Yaskawa INFORM job: apremTRJ1.JBI

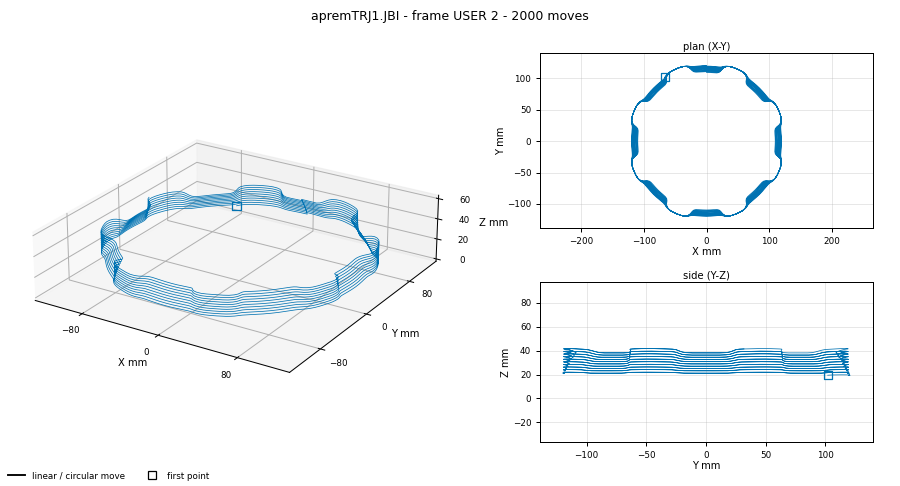
[picture p0: tool path of apremTRJ1.JBI in frame USER 2, 2000 of 2000 moves have a stored position in this frame; points joined in program order, loops and branches not executed]
/JOB
//NAME apremTRJ1
//POS
///NPOS 2000,0,0,0,0,0
///USER 2
///TOOL 1
///POSTYPE USER
///RECTAN
///RCONF 1,0,0,0,0,0,0,0,0,0,0,0,0,0,0,0,0,0,0,0,0,0,0,0
C00000=-66.629,101.942,19.455,-170.1157,12.4530,0.0000
C00001=-65.347,103.638,19.586,-173.5152,9.1234,0.0000
C00002=-64.038,105.345,19.680,-175.2675,5.6483,0.0000
C00003=-62.177,107.232,19.725,-176.7314,2.8984,0.0000
C00004=-59.447,109.388,19.749,-178.4360,1.1171,0.0000
C00005=-56.168,111.510,19.767,-179.6465,0.2072,0.0000
C00006=-52.762,113.295,19.786,-179.9247,0.0358,0.0000
C00007=-49.468,114.792,19.798,-179.9913,0.0038,0.0000
C00008=-46.191,116.149,19.798,-179.9912,0.0035,0.0000
C00009=-42.803,117.420,19.786,-179.9215,0.0280,0.0000
C00010=-39.133,118.567,19.767,-179.6035,0.1035,0.0000
C00011=-35.314,119.384,19.749,-178.1045,0.3162,0.0000
C00012=-31.859,119.791,19.725,-175.6434,0.2625,0.0000
C00013=-29.209,119.772,19.680,-172.6791,-0.6529,0.0000
C00014=-27.076,119.491,19.586,-169.0248,-1.9005,0.0000
C00015=-24.970,119.198,19.455,-164.3916,-1.8868,0.0000
C00016=-22.390,119.093,19.319,-160.1217,-0.0530,0.0000
C00017=-18.637,119.331,19.213,-157.6149,2.1562,0.0000
C00018=-13.062,119.916,19.170,-156.7679,2.4486,0.0000
C00019=-6.840,120.423,19.168,-156.6463,1.4246,0.0000
C00020=0.000,120.619,19.169,-156.6224,0.0002,0.0000
C00021=0.000,119.715,21.175,-154.8867,0.0002,0.0000
C00022=6.757,119.522,21.173,-154.9119,-1.5414,0.0000
C00023=12.923,119.024,21.176,-155.0380,-2.5924,0.0000
C00024=18.467,118.472,21.232,-155.9401,-1.9735,0.0000
C00025=22.185,118.320,21.368,-158.8454,1.0092,0.0000
C00026=24.738,118.553,21.546,-163.9075,3.1512,0.0000
C00027=26.827,119.004,21.717,-169.0787,2.8689,0.0000
C00028=28.944,119.457,21.842,-172.7347,1.2029,0.0000
C00029=31.572,119.635,21.901,-175.6219,-0.0566,0.0000
C00030=35.044,119.351,21.932,-178.1277,-0.2593,0.0000
C00031=38.919,118.606,21.957,-179.6493,-0.0862,0.0000
C00032=42.669,117.464,21.982,-179.9232,-0.0272,0.0000
C00033=46.146,116.167,21.998,-179.9915,-0.0033,0.0000
C00034=49.513,114.773,21.998,-179.9916,-0.0037,0.0000
C00035=52.889,113.231,21.982,-179.9265,-0.0351,0.0000
C00036=56.347,111.387,21.957,-179.6910,-0.1870,0.0000
C00037=59.614,109.174,21.932,-178.4926,-1.1409,0.0000
C00038=62.270,106.919,21.901,-176.8613,-3.0589,0.0000
C00039=64.002,104.935,21.842,-175.6938,-5.9938,0.0000
C00040=65.179,103.118,21.717,-174.2325,-9.7524,0.0000
C00041=66.337,101.322,21.546,-170.6269,-13.6541,0.0000
C00042=67.977,99.352,21.368,-165.3631,-15.9648,0.0000
C00043=70.714,96.831,21.232,-161.2181,-16.2433,0.0000
C00044=75.024,93.301,21.176,-160.1416,-16.5489,0.0000
C00045=79.737,89.293,21.173,-160.7058,-17.3293,0.0000
C00046=84.652,84.652,21.175,-161.6632,-18.3371,0.0000
C00047=89.293,79.737,21.173,-162.6706,-19.2941,0.0000
C00048=93.301,75.024,21.176,-163.4508,-19.8582,0.0000
C00049=96.831,70.714,21.232,-163.7569,-18.7820,0.0000
C00050=99.352,67.977,21.368,-164.0352,-14.6369,0.0000
C00051=101.322,66.337,21.546,-166.3459,-9.3731,0.0000
C00052=103.118,65.179,21.717,-170.2476,-5.7675,0.0000
C00053=104.935,64.002,21.842,-174.0062,-4.3062,0.0000
C00054=106.919,62.270,21.901,-176.9411,-3.1387,0.0000
C00055=109.174,59.614,21.932,-178.8591,-1.5074,0.0000
C00056=111.387,56.347,21.957,-179.8130,-0.3090,0.0000
C00057=113.231,52.889,21.982,-179.9649,-0.0735,0.0000
C00058=114.773,49.513,21.998,-179.9963,-0.0084,0.0000
C00059=116.167,46.146,21.998,-179.9967,-0.0085,0.0000
C00060=117.464,42.669,21.982,-179.9728,-0.0768,0.0000
C00061=118.606,38.919,21.957,-179.9138,-0.3507,0.0000
C00062=119.351,35.044,21.932,-179.7407,-1.8723,0.0000
C00063=119.635,31.572,21.901,-179.9434,-4.3781,0.0000
C00064=119.457,28.944,21.842,178.7971,-7.2653,0.0000
C00065=119.004,26.827,21.717,177.1311,-10.9213,0.0000
C00066=118.553,24.738,21.546,176.8488,-16.0925,0.0000
C00067=118.320,22.185,21.368,178.9908,-21.1546,0.0000
C00068=118.472,18.467,21.232,-178.0265,-24.0599,0.0000
C00069=119.024,12.923,21.176,-177.4076,-24.9620,0.0000
C00070=119.522,6.757,21.173,-178.4586,-25.0881,0.0000
C00071=119.715,0.000,21.175,179.9998,-25.1133,0.0000
C00072=119.522,-6.757,21.173,178.4588,-25.0881,0.0000
C00073=119.024,-12.923,21.176,177.4079,-24.9620,0.0000
C00074=118.472,-18.468,21.232,178.0263,-24.0599,0.0000
C00075=118.320,-22.185,21.368,-178.9908,-21.1546,0.0000
C00076=118.553,-24.738,21.546,-176.8488,-16.0925,0.0000
C00077=119.004,-26.827,21.717,-177.1311,-10.9213,0.0000
C00078=119.457,-28.944,21.842,-178.7971,-7.2653,0.0000
C00079=119.635,-31.572,21.901,179.9434,-4.3781,0.0000
C00080=119.351,-35.044,21.932,179.7407,-1.8723,0.0000
C00081=118.606,-38.919,21.957,179.9138,-0.3507,0.0000
C00082=117.464,-42.669,21.982,179.9728,-0.0768,0.0000
C00083=116.167,-46.146,21.998,179.9967,-0.0085,0.0000
C00084=114.773,-49.513,21.998,179.9963,-0.0084,0.0000
C00085=113.231,-52.889,21.982,179.9649,-0.0735,0.0000
C00086=111.387,-56.347,21.957,179.8130,-0.3090,0.0000
C00087=109.174,-59.614,21.932,178.8591,-1.5074,0.0000
C00088=106.919,-62.270,21.901,176.9411,-3.1387,0.0000
C00089=104.935,-64.002,21.842,174.0062,-4.3062,0.0000
C00090=103.118,-65.179,21.717,170.2476,-5.7675,0.0000
C00091=101.322,-66.337,21.546,166.3459,-9.3731,0.0000
C00092=99.352,-67.977,21.368,164.0352,-14.6369,0.0000
C00093=96.831,-70.714,21.232,163.7567,-18.7819,0.0000
C00094=93.301,-75.024,21.176,163.4511,-19.8584,0.0000
C00095=89.293,-79.737,21.173,162.6707,-19.2942,0.0000
C00096=84.652,-84.652,21.175,161.6629,-18.3368,0.0000
C00097=79.737,-89.293,21.173,160.7059,-17.3294,0.0000
C00098=75.024,-93.301,21.176,160.1418,-16.5492,0.0000
C00099=70.714,-96.831,21.232,161.2180,-16.2431,0.0000
C00100=67.977,-99.352,21.368,165.3631,-15.9648,0.0000
C00101=66.337,-101.322,21.546,170.6269,-13.6541,0.0000
C00102=65.179,-103.118,21.717,174.2325,-9.7524,0.0000
C00103=64.002,-104.935,21.842,175.6938,-5.9938,0.0000
C00104=62.270,-106.919,21.901,176.8613,-3.0589,0.0000
C00105=59.614,-109.174,21.932,178.4926,-1.1409,0.0000
C00106=56.347,-111.387,21.957,179.6910,-0.1870,0.0000
C00107=52.889,-113.231,21.982,179.9265,-0.0351,0.0000
C00108=49.513,-114.773,21.998,179.9916,-0.0037,0.0000
C00109=46.146,-116.167,21.998,179.9915,-0.0033,0.0000
C00110=42.669,-117.464,21.982,179.9232,-0.0272,0.0000
C00111=38.919,-118.606,21.957,179.6493,-0.0862,0.0000
C00112=35.044,-119.351,21.932,178.1277,-0.2593,0.0000
C00113=31.572,-119.635,21.901,175.6219,-0.0566,0.0000
C00114=28.944,-119.457,21.842,172.7347,1.2029,0.0000
C00115=26.827,-119.004,21.717,169.0787,2.8689,0.0000
C00116=24.738,-118.553,21.546,163.9075,3.1512,0.0000
C00117=22.185,-118.320,21.368,158.8454,1.0092,0.0000
C00118=18.467,-118.472,21.232,155.9401,-1.9735,0.0000
C00119=12.923,-119.024,21.176,155.0380,-2.5924,0.0000
C00120=6.757,-119.522,21.173,154.9119,-1.5414,0.0000
C00121=0.000,-119.715,21.175,154.8867,0.0002,0.0000
C00122=0.000,-119.715,21.175,154.8867,0.0002,0.0000
C00123=-6.757,-119.522,21.173,154.9119,1.5412,0.0000
C00124=-12.923,-119.024,21.176,155.0380,2.5921,0.0000
C00125=-18.468,-118.472,21.232,155.9401,1.9737,0.0000
C00126=-22.185,-118.320,21.368,158.8454,-1.0092,0.0000
C00127=-24.738,-118.553,21.546,163.9075,-3.1512,0.0000
C00128=-26.827,-119.004,21.717,169.0787,-2.8689,0.0000
C00129=-28.944,-119.457,21.842,172.7347,-1.2029,0.0000
C00130=-31.572,-119.635,21.901,175.6219,0.0566,0.0000
C00131=-35.044,-119.351,21.932,178.1277,0.2593,0.0000
C00132=-38.919,-118.606,21.957,179.6493,0.0862,0.0000
C00133=-42.669,-117.464,21.982,179.9232,0.0272,0.0000
C00134=-46.146,-116.167,21.998,179.9915,0.0033,0.0000
C00135=-49.513,-114.773,21.998,179.9916,0.0037,0.0000
C00136=-52.889,-113.231,21.982,179.9265,0.0351,0.0000
C00137=-56.347,-111.387,21.957,179.6910,0.1870,0.0000
C00138=-59.614,-109.174,21.932,178.4926,1.1409,0.0000
C00139=-62.270,-106.919,21.901,176.8613,3.0589,0.0000
C00140=-64.002,-104.935,21.842,175.6938,5.9938,0.0000
C00141=-65.179,-103.118,21.717,174.2325,9.7524,0.0000
C00142=-66.337,-101.322,21.546,170.6269,13.6541,0.0000
C00143=-67.977,-99.352,21.368,165.3631,15.9648,0.0000
C00144=-70.714,-96.831,21.232,161.2181,16.2433,0.0000
C00145=-75.024,-93.301,21.176,160.1416,16.5489,0.0000
C00146=-79.737,-89.293,21.173,160.7058,17.3293,0.0000
C00147=-84.652,-84.652,21.175,161.6632,18.3371,0.0000
C00148=-89.293,-79.737,21.173,162.6706,19.2941,0.0000
C00149=-93.301,-75.024,21.176,163.4508,19.8582,0.0000
C00150=-96.831,-70.714,21.232,163.7569,18.7820,0.0000
C00151=-99.352,-67.977,21.368,164.0352,14.6369,0.0000
C00152=-101.322,-66.337,21.546,166.3459,9.3731,0.0000
C00153=-103.118,-65.179,21.717,170.2476,5.7675,0.0000
C00154=-104.935,-64.002,21.842,174.0062,4.3062,0.0000
C00155=-106.919,-62.270,21.901,176.9411,3.1387,0.0000
C00156=-109.174,-59.614,21.932,178.8591,1.5074,0.0000
C00157=-111.387,-56.347,21.957,179.8130,0.3090,0.0000
C00158=-113.231,-52.889,21.982,179.9649,0.0735,0.0000
C00159=-114.773,-49.513,21.998,179.9963,0.0084,0.0000
C00160=-116.167,-46.146,21.998,179.9967,0.0085,0.0000
C00161=-117.464,-42.669,21.982,179.9728,0.0768,0.0000
C00162=-118.606,-38.919,21.957,179.9138,0.3507,0.0000
C00163=-119.351,-35.044,21.932,179.7407,1.8723,0.0000
C00164=-119.635,-31.572,21.901,179.9434,4.3781,0.0000
C00165=-119.457,-28.944,21.842,-178.7971,7.2653,0.0000
C00166=-119.004,-26.827,21.717,-177.1311,10.9213,0.0000
C00167=-118.553,-24.738,21.546,-176.8488,16.0925,0.0000
C00168=-118.320,-22.185,21.368,-178.9908,21.1546,0.0000
C00169=-118.472,-18.467,21.232,178.0265,24.0599,0.0000
C00170=-119.024,-12.923,21.176,177.4076,24.9620,0.0000
C00171=-119.522,-6.757,21.173,178.4586,25.0881,0.0000
C00172=-119.715,0.000,21.175,-179.9998,25.1133,0.0000
C00173=-119.522,6.757,21.173,-178.4588,25.0881,0.0000
C00174=-119.024,12.923,21.176,-177.4079,24.9620,0.0000
C00175=-118.472,18.468,21.232,-178.0263,24.0599,0.0000
C00176=-118.320,22.185,21.368,178.9908,21.1546,0.0000
C00177=-118.553,24.738,21.546,176.8488,16.0925,0.0000
C00178=-119.004,26.827,21.717,177.1311,10.9213,0.0000
C00179=-119.457,28.944,21.842,178.7971,7.2653,0.0000
C00180=-119.635,31.572,21.901,-179.9434,4.3781,0.0000
C00181=-119.351,35.044,21.932,-179.7407,1.8723,0.0000
C00182=-118.606,38.919,21.957,-179.9138,0.3507,0.0000
C00183=-117.464,42.669,21.982,-179.9728,0.0768,0.0000
C00184=-116.167,46.146,21.998,-179.9967,0.0085,0.0000
C00185=-114.773,49.513,21.998,-179.9963,0.0084,0.0000
C00186=-113.231,52.889,21.982,-179.9649,0.0735,0.0000
C00187=-111.387,56.347,21.957,-179.8130,0.3090,0.0000
C00188=-109.174,59.614,21.932,-178.8591,1.5074,0.0000
C00189=-106.919,62.270,21.901,-176.9411,3.1387,0.0000
C00190=-104.935,64.002,21.842,-174.0062,4.3062,0.0000
C00191=-103.118,65.179,21.717,-170.2476,5.7675,0.0000
C00192=-101.322,66.337,21.546,-166.3459,9.3731,0.0000
C00193=-99.352,67.977,21.368,-164.0352,14.6369,0.0000
C00194=-96.831,70.714,21.232,-163.7567,18.7819,0.0000
C00195=-93.301,75.024,21.176,-163.4511,19.8584,0.0000
C00196=-89.293,79.737,21.173,-162.6707,19.2942,0.0000
C00197=-84.652,84.652,21.175,-161.6629,18.3368,0.0000
C00198=-79.737,89.293,21.173,-160.7059,17.3294,0.0000
C00199=-75.024,93.301,21.176,-160.1418,16.5492,0.0000
C00200=-70.714,96.831,21.232,-161.2180,16.2431,0.0000
C00201=-67.977,99.352,21.368,-165.3631,15.9648,0.0000
C00202=-66.337,101.322,21.546,-170.6269,13.6541,0.0000
C00203=-65.179,103.118,21.717,-174.2325,9.7524,0.0000
C00204=-64.002,104.935,21.842,-175.6938,5.9938,0.0000
C00205=-62.270,106.919,21.901,-176.8613,3.0589,0.0000
C00206=-59.614,109.174,21.932,-178.4926,1.1409,0.0000
C00207=-56.347,111.387,21.957,-179.6910,0.1870,0.0000
C00208=-52.889,113.231,21.982,-179.9265,0.0351,0.0000
C00209=-49.513,114.773,21.998,-179.9916,0.0037,0.0000
C00210=-46.146,116.167,21.998,-179.9915,0.0033,0.0000
C00211=-42.669,117.464,21.982,-179.9232,0.0272,0.0000
C00212=-38.919,118.606,21.957,-179.6493,0.0862,0.0000
C00213=-35.044,119.351,21.932,-178.1277,0.2593,0.0000
C00214=-31.572,119.635,21.901,-175.6219,0.0566,0.0000
C00215=-28.944,119.457,21.842,-172.7347,-1.2029,0.0000
C00216=-26.827,119.004,21.717,-169.0787,-2.8689,0.0000
C00217=-24.738,118.553,21.546,-163.9075,-3.1512,0.0000
C00218=-22.185,118.320,21.368,-158.8454,-1.0092,0.0000
C00219=-18.468,118.472,21.232,-155.9401,1.9737,0.0000
C00220=-12.923,119.024,21.176,-155.0380,2.5921,0.0000
C00221=-6.757,119.522,21.173,-154.9119,1.5412,0.0000
C00222=0.000,119.715,21.175,-154.8867,0.0002,0.0000
C00223=0.000,118.754,23.154,-153.2988,0.0002,0.0000
C00224=6.669,118.564,23.151,-153.3252,-1.6500,0.0000
C00225=12.776,118.074,23.155,-153.4547,-2.7089,0.0000
C00226=18.287,117.558,23.225,-154.4168,-1.6956,0.0000
C00227=21.966,117.495,23.396,-157.8261,2.1572,0.0000
C00228=24.490,117.863,23.620,-163.8200,4.4801,0.0000
C00229=26.560,118.482,23.837,-169.5033,3.7726,0.0000
C00230=28.658,119.117,23.996,-173.0515,1.7294,0.0000
C00231=31.262,119.466,24.073,-175.7313,0.1639,0.0000
C00232=34.753,119.316,24.112,-178.2061,-0.1949,0.0000
C00233=38.689,118.647,24.144,-179.7139,-0.0658,0.0000
C00234=42.523,117.512,24.176,-179.9268,-0.0257,0.0000
C00235=46.096,116.186,24.197,-179.9920,-0.0031,0.0000
C00236=49.561,114.751,24.197,-179.9921,-0.0034,0.0000
C00237=53.026,113.162,24.176,-179.9301,-0.0336,0.0000
C00238=56.539,111.253,24.144,-179.7511,-0.1558,0.0000
C00239=59.796,108.943,24.112,-178.5936,-1.1309,0.0000
C00240=62.370,106.581,24.073,-177.0944,-3.1368,0.0000
C00241=63.964,104.493,23.996,-176.2909,-6.1372,0.0000
C00242=64.998,102.560,23.837,-175.1764,-10.0729,0.0000
C00243=66.025,100.658,23.620,-171.4825,-14.6048,0.0000
C00244=67.549,98.614,23.396,-165.3424,-17.4753,0.0000
C00245=70.195,96.057,23.225,-160.2282,-17.6199,0.0000
C00246=74.457,92.525,23.155,-158.8582,-17.7339,0.0000
C00247=79.121,88.553,23.151,-159.4130,-18.5146,0.0000
C00248=83.972,83.972,23.154,-160.4219,-19.5784,0.0000
C00249=88.553,79.121,23.151,-161.4852,-20.5868,0.0000
C00250=92.525,74.457,23.155,-162.2659,-21.1415,0.0000
C00251=96.057,70.195,23.225,-162.3803,-19.7719,0.0000
C00252=98.614,67.549,23.396,-162.5247,-14.6576,0.0000
C00253=100.658,66.025,23.620,-165.3952,-8.5175,0.0000
C00254=102.560,64.998,23.837,-169.9271,-4.8236,0.0000
C00255=104.493,63.964,23.996,-173.8628,-3.7091,0.0000
C00256=106.581,62.370,24.073,-176.8632,-2.9056,0.0000
C00257=108.943,59.796,24.112,-178.8691,-1.4064,0.0000
C00258=111.253,56.539,24.144,-179.8442,-0.2489,0.0000
C00259=113.162,53.026,24.176,-179.9664,-0.0699,0.0000
C00260=114.751,49.561,24.197,-179.9966,-0.0079,0.0000
C00261=116.186,46.096,24.197,-179.9969,-0.0080,0.0000
C00262=117.512,42.523,24.176,-179.9743,-0.0732,0.0000
C00263=118.647,38.689,24.144,-179.9342,-0.2861,0.0000
C00264=119.316,34.753,24.112,-179.8051,-1.7939,0.0000
C00265=119.466,31.262,24.073,179.8361,-4.2687,0.0000
C00266=119.117,28.658,23.996,178.2706,-6.9485,0.0000
C00267=118.482,26.560,23.837,176.2274,-10.4967,0.0000
C00268=117.863,24.490,23.620,175.5199,-16.1800,0.0000
C00269=117.495,21.966,23.396,177.8428,-22.1739,0.0000
C00270=117.558,18.287,23.225,-178.3044,-25.5832,0.0000
C00271=118.074,12.776,23.155,-177.2911,-26.5453,0.0000
C00272=118.564,6.669,23.151,-178.3500,-26.6748,0.0000
C00273=118.754,0.000,23.154,179.9998,-26.7012,0.0000
C00274=118.564,-6.669,23.151,178.3503,-26.6748,0.0000
C00275=118.074,-12.776,23.155,177.2915,-26.5453,0.0000
C00276=117.558,-18.287,23.225,178.3041,-25.5831,0.0000
C00277=117.495,-21.966,23.396,-177.8428,-22.1739,0.0000
C00278=117.863,-24.490,23.620,-175.5199,-16.1800,0.0000
C00279=118.482,-26.560,23.837,-176.2274,-10.4967,0.0000
C00280=119.117,-28.658,23.996,-178.2706,-6.9485,0.0000
C00281=119.466,-31.262,24.073,-179.8361,-4.2687,0.0000
C00282=119.316,-34.753,24.112,179.8051,-1.7939,0.0000
C00283=118.647,-38.689,24.144,179.9342,-0.2861,0.0000
C00284=117.512,-42.523,24.176,179.9743,-0.0732,0.0000
C00285=116.186,-46.096,24.197,179.9969,-0.0080,0.0000
C00286=114.751,-49.561,24.197,179.9966,-0.0079,0.0000
C00287=113.162,-53.026,24.176,179.9664,-0.0699,0.0000
C00288=111.253,-56.539,24.144,179.8442,-0.2489,0.0000
C00289=108.943,-59.796,24.112,178.8691,-1.4064,0.0000
C00290=106.581,-62.370,24.073,176.8632,-2.9056,0.0000
C00291=104.493,-63.964,23.996,173.8628,-3.7091,0.0000
C00292=102.560,-64.998,23.837,169.9271,-4.8236,0.0000
C00293=100.658,-66.025,23.620,165.3952,-8.5175,0.0000
C00294=98.614,-67.549,23.396,162.5247,-14.6576,0.0000
C00295=96.057,-70.195,23.225,162.3801,-19.7718,0.0000
C00296=92.525,-74.457,23.155,162.2661,-21.1418,0.0000
C00297=88.553,-79.121,23.151,161.4854,-20.5870,0.0000
C00298=83.972,-83.972,23.154,160.4216,-19.5781,0.0000
C00299=79.121,-88.553,23.151,159.4132,-18.5148,0.0000
C00300=74.457,-92.525,23.155,158.8585,-17.7341,0.0000
C00301=70.195,-96.057,23.225,160.2281,-17.6197,0.0000
C00302=67.549,-98.614,23.396,165.3424,-17.4753,0.0000
C00303=66.025,-100.658,23.620,171.4825,-14.6048,0.0000
C00304=64.998,-102.560,23.837,175.1764,-10.0729,0.0000
C00305=63.964,-104.493,23.996,176.2909,-6.1372,0.0000
C00306=62.370,-106.581,24.073,177.0944,-3.1368,0.0000
C00307=59.796,-108.943,24.112,178.5936,-1.1309,0.0000
C00308=56.539,-111.253,24.144,179.7511,-0.1558,0.0000
C00309=53.026,-113.162,24.176,179.9301,-0.0336,0.0000
C00310=49.561,-114.751,24.197,179.9921,-0.0034,0.0000
C00311=46.096,-116.186,24.197,179.9920,-0.0031,0.0000
C00312=42.523,-117.512,24.176,179.9268,-0.0257,0.0000
C00313=38.689,-118.647,24.144,179.7139,-0.0658,0.0000
C00314=34.753,-119.316,24.112,178.2061,-0.1949,0.0000
C00315=31.262,-119.466,24.073,175.7313,0.1639,0.0000
C00316=28.658,-119.117,23.996,173.0515,1.7294,0.0000
C00317=26.560,-118.482,23.837,169.5033,3.7726,0.0000
C00318=24.490,-117.863,23.620,163.8200,4.4801,0.0000
C00319=21.966,-117.495,23.396,157.8261,2.1572,0.0000
C00320=18.287,-117.558,23.225,154.4168,-1.6956,0.0000
C00321=12.776,-118.074,23.155,153.4547,-2.7089,0.0000
C00322=6.669,-118.564,23.151,153.3252,-1.6500,0.0000
C00323=0.000,-118.754,23.154,153.2988,0.0002,0.0000
C00324=0.000,-118.754,23.154,153.2988,0.0002,0.0000
C00325=-6.669,-118.564,23.151,153.3252,1.6497,0.0000
C00326=-12.776,-118.074,23.155,153.4547,2.7085,0.0000
C00327=-18.287,-117.558,23.225,154.4169,1.6959,0.0000
C00328=-21.966,-117.495,23.396,157.8261,-2.1572,0.0000
C00329=-24.490,-117.863,23.620,163.8200,-4.4801,0.0000
C00330=-26.560,-118.482,23.837,169.5033,-3.7726,0.0000
C00331=-28.658,-119.117,23.996,173.0515,-1.7294,0.0000
C00332=-31.262,-119.466,24.073,175.7313,-0.1639,0.0000
C00333=-34.753,-119.316,24.112,178.2061,0.1949,0.0000
C00334=-38.689,-118.647,24.144,179.7139,0.0658,0.0000
C00335=-42.523,-117.512,24.176,179.9268,0.0257,0.0000
C00336=-46.096,-116.186,24.197,179.9920,0.0031,0.0000
C00337=-49.561,-114.751,24.197,179.9921,0.0034,0.0000
C00338=-53.026,-113.162,24.176,179.9301,0.0336,0.0000
C00339=-56.539,-111.253,24.144,179.7511,0.1558,0.0000
C00340=-59.796,-108.943,24.112,178.5936,1.1309,0.0000
C00341=-62.370,-106.581,24.073,177.0944,3.1368,0.0000
C00342=-63.964,-104.493,23.996,176.2909,6.1372,0.0000
C00343=-64.998,-102.560,23.837,175.1764,10.0729,0.0000
C00344=-66.025,-100.658,23.620,171.4825,14.6048,0.0000
C00345=-67.549,-98.614,23.396,165.3424,17.4753,0.0000
C00346=-70.195,-96.057,23.225,160.2282,17.6199,0.0000
C00347=-74.457,-92.525,23.155,158.8582,17.7339,0.0000
C00348=-79.121,-88.553,23.151,159.4130,18.5146,0.0000
C00349=-83.972,-83.972,23.154,160.4219,19.5784,0.0000
C00350=-88.553,-79.121,23.151,161.4852,20.5868,0.0000
C00351=-92.525,-74.457,23.155,162.2659,21.1415,0.0000
C00352=-96.057,-70.195,23.225,162.3803,19.7719,0.0000
C00353=-98.614,-67.549,23.396,162.5247,14.6576,0.0000
C00354=-100.658,-66.025,23.620,165.3952,8.5175,0.0000
C00355=-102.560,-64.998,23.837,169.9271,4.8236,0.0000
C00356=-104.493,-63.964,23.996,173.8628,3.7091,0.0000
C00357=-106.581,-62.370,24.073,176.8632,2.9056,0.0000
C00358=-108.943,-59.796,24.112,178.8691,1.4064,0.0000
C00359=-111.253,-56.539,24.144,179.8442,0.2489,0.0000
C00360=-113.162,-53.026,24.176,179.9664,0.0699,0.0000
C00361=-114.751,-49.561,24.197,179.9966,0.0079,0.0000
C00362=-116.186,-46.096,24.197,179.9969,0.0080,0.0000
C00363=-117.512,-42.523,24.176,179.9743,0.0732,0.0000
C00364=-118.647,-38.689,24.144,179.9342,0.2861,0.0000
C00365=-119.316,-34.753,24.112,179.8051,1.7939,0.0000
C00366=-119.466,-31.262,24.073,-179.8361,4.2687,0.0000
C00367=-119.117,-28.658,23.996,-178.2706,6.9485,0.0000
C00368=-118.482,-26.560,23.837,-176.2274,10.4967,0.0000
C00369=-117.863,-24.490,23.620,-175.5199,16.1800,0.0000
C00370=-117.495,-21.966,23.396,-177.8428,22.1739,0.0000
C00371=-117.558,-18.287,23.225,178.3044,25.5832,0.0000
C00372=-118.074,-12.776,23.155,177.2911,26.5453,0.0000
C00373=-118.564,-6.669,23.151,178.3500,26.6748,0.0000
C00374=-118.754,0.000,23.154,-179.9998,26.7012,0.0000
C00375=-118.564,6.669,23.151,-178.3503,26.6748,0.0000
C00376=-118.074,12.776,23.155,-177.2915,26.5453,0.0000
C00377=-117.558,18.287,23.225,-178.3041,25.5831,0.0000
C00378=-117.495,21.966,23.396,177.8428,22.1739,0.0000
C00379=-117.863,24.490,23.620,175.5199,16.1800,0.0000
C00380=-118.482,26.560,23.837,176.2274,10.4967,0.0000
C00381=-119.117,28.658,23.996,178.2706,6.9485,0.0000
C00382=-119.466,31.262,24.073,179.8361,4.2687,0.0000
C00383=-119.316,34.753,24.112,-179.8051,1.7939,0.0000
C00384=-118.647,38.689,24.144,-179.9342,0.2861,0.0000
C00385=-117.512,42.523,24.176,-179.9743,0.0732,0.0000
C00386=-116.186,46.096,24.197,-179.9969,0.0080,0.0000
C00387=-114.751,49.561,24.197,-179.9966,0.0079,0.0000
C00388=-113.162,53.026,24.176,-179.9664,0.0699,0.0000
C00389=-111.253,56.539,24.144,-179.8442,0.2489,0.0000
C00390=-108.943,59.796,24.112,-178.8691,1.4064,0.0000
C00391=-106.581,62.370,24.073,-176.8632,2.9056,0.0000
C00392=-104.493,63.964,23.996,-173.8628,3.7091,0.0000
C00393=-102.560,64.998,23.837,-169.9271,4.8236,0.0000
C00394=-100.658,66.025,23.620,-165.3952,8.5175,0.0000
C00395=-98.614,67.549,23.396,-162.5247,14.6576,0.0000
C00396=-96.057,70.195,23.225,-162.3801,19.7718,0.0000
C00397=-92.525,74.457,23.155,-162.2661,21.1418,0.0000
C00398=-88.553,79.121,23.151,-161.4854,20.5870,0.0000
C00399=-83.972,83.972,23.154,-160.4216,19.5781,0.0000
C00400=-79.121,88.553,23.151,-159.4132,18.5148,0.0000
C00401=-74.457,92.525,23.155,-158.8585,17.7341,0.0000
C00402=-70.195,96.057,23.225,-160.2281,17.6197,0.0000
C00403=-67.549,98.614,23.396,-165.3424,17.4753,0.0000
C00404=-66.025,100.658,23.620,-171.4825,14.6048,0.0000
C00405=-64.998,102.560,23.837,-175.1764,10.0729,0.0000
C00406=-63.964,104.493,23.996,-176.2909,6.1372,0.0000
C00407=-62.370,106.581,24.073,-177.0944,3.1368,0.0000
C00408=-59.796,108.943,24.112,-178.5936,1.1309,0.0000
C00409=-56.539,111.253,24.144,-179.7511,0.1558,0.0000
C00410=-53.026,113.162,24.176,-179.9301,0.0336,0.0000
C00411=-49.561,114.751,24.197,-179.9921,0.0034,0.0000
C00412=-46.096,116.186,24.197,-179.9920,0.0031,0.0000
C00413=-42.523,117.512,24.176,-179.9268,0.0257,0.0000
C00414=-38.689,118.647,24.144,-179.7139,0.0658,0.0000
C00415=-34.753,119.316,24.112,-178.2061,0.1949,0.0000
C00416=-31.262,119.466,24.073,-175.7313,-0.1639,0.0000
C00417=-28.658,119.117,23.996,-173.0515,-1.7294,0.0000
C00418=-26.560,118.482,23.837,-169.5033,-3.7726,0.0000
C00419=-24.490,117.863,23.620,-163.8200,-4.4801,0.0000
C00420=-21.966,117.495,23.396,-157.8261,-2.1572,0.0000
C00421=-18.287,117.558,23.225,-154.4169,1.6959,0.0000
C00422=-12.776,118.074,23.155,-153.4547,2.7085,0.0000
C00423=-6.669,118.564,23.151,-153.3252,1.6497,0.0000
C00424=0.000,118.754,23.154,-153.2988,0.0002,0.0000
C00425=0.000,117.740,25.106,-151.8484,0.0003,0.0000
C00426=6.577,117.553,25.104,-151.8757,-1.7507,0.0000
C00427=12.620,117.073,25.107,-152.0079,-2.7988,0.0000
C00428=18.097,116.593,25.193,-153.0392,-1.3238,0.0000
C00429=21.735,116.622,25.402,-157.0835,3.4645,0.0000
C00430=24.226,117.130,25.677,-164.1300,5.7683,0.0000
C00431=26.275,117.926,25.947,-170.2564,4.5098,0.0000
C00432=28.354,118.754,26.145,-173.6147,2.1641,0.0000
C00433=30.931,119.286,26.240,-175.9744,0.3765,0.0000
C00434=34.441,119.279,26.290,-178.3387,-0.1287,0.0000
C00435=38.442,118.692,26.330,-179.7962,-0.0436,0.0000
C00436=42.367,117.564,26.370,-179.9323,-0.0236,0.0000
C00437=46.044,116.206,26.396,-179.9928,-0.0028,0.0000
C00438=49.613,114.728,26.396,-179.9929,-0.0031,0.0000
C00439=53.172,113.088,26.370,-179.9354,-0.0312,0.0000
C00440=56.745,111.111,26.330,-179.8251,-0.1133,0.0000
C00441=59.989,108.697,26.290,-178.7342,-1.0839,0.0000
C00442=62.476,106.220,26.240,-177.4167,-3.1144,0.0000
C00443=63.923,104.021,26.145,-176.9999,-6.0423,0.0000
C00444=64.806,101.965,25.947,-176.2439,-10.0482,0.0000
C00445=65.693,99.954,25.677,-172.6160,-15.2406,0.0000
C00446=67.095,97.833,25.402,-165.6340,-18.8675,0.0000
C00447=69.647,95.240,25.193,-159.3927,-18.9494,0.0000
C00448=73.859,91.707,25.107,-157.6858,-18.8439,0.0000
C00449=78.472,87.773,25.104,-158.2204,-19.6126,0.0000
C00450=83.255,83.255,25.106,-159.2746,-20.7257,0.0000
C00451=87.773,78.472,25.104,-160.3872,-21.7793,0.0000
C00452=91.707,73.859,25.107,-161.1558,-22.3139,0.0000
C00453=95.240,69.647,25.193,-161.0509,-20.6075,0.0000
C00454=97.833,67.095,25.402,-161.1325,-14.3660,0.0000
C00455=99.954,65.693,25.677,-164.7594,-7.3840,0.0000
C00456=101.965,64.806,25.947,-169.9518,-3.7561,0.0000
C00457=104.021,63.923,26.145,-173.9577,-3.0001,0.0000
C00458=106.220,62.476,26.240,-176.8856,-2.5833,0.0000
C00459=108.697,59.989,26.290,-178.9161,-1.2658,0.0000
C00460=111.111,56.745,26.330,-179.8867,-0.1749,0.0000
C00461=113.088,53.172,26.370,-179.9688,-0.0646,0.0000
C00462=114.728,49.613,26.396,-179.9969,-0.0071,0.0000
C00463=116.206,46.044,26.396,-179.9972,-0.0072,0.0000
C00464=117.564,42.367,26.370,-179.9764,-0.0677,0.0000
C00465=118.692,38.442,26.330,-179.9564,-0.2038,0.0000
C00466=119.279,34.441,26.290,-179.8713,-1.6613,0.0000
C00467=119.286,30.931,26.240,179.6235,-4.0256,0.0000
C00468=118.754,28.354,26.145,177.8359,-6.3853,0.0000
C00469=117.926,26.275,25.947,175.4902,-9.7436,0.0000
C00470=117.130,24.226,25.677,174.2317,-15.8700,0.0000
C00471=116.622,21.735,25.402,176.5355,-22.9165,0.0000
C00472=116.593,18.097,25.193,-178.6762,-26.9608,0.0000
C00473=117.073,12.620,25.107,-177.2012,-27.9921,0.0000
C00474=117.553,6.577,25.104,-178.2493,-28.1243,0.0000
C00475=117.740,0.000,25.106,179.9997,-28.1516,0.0000
C00476=117.553,-6.577,25.104,178.2496,-28.1243,0.0000
C00477=117.073,-12.620,25.107,177.2017,-27.9921,0.0000
C00478=116.593,-18.097,25.193,178.6758,-26.9608,0.0000
C00479=116.622,-21.735,25.402,-176.5355,-22.9165,0.0000
C00480=117.130,-24.226,25.677,-174.2317,-15.8700,0.0000
C00481=117.926,-26.275,25.947,-175.4902,-9.7436,0.0000
C00482=118.754,-28.354,26.145,-177.8359,-6.3853,0.0000
C00483=119.286,-30.931,26.240,-179.6235,-4.0256,0.0000
C00484=119.279,-34.441,26.290,179.8713,-1.6613,0.0000
C00485=118.692,-38.442,26.330,179.9564,-0.2038,0.0000
C00486=117.564,-42.367,26.370,179.9764,-0.0677,0.0000
C00487=116.206,-46.044,26.396,179.9972,-0.0072,0.0000
C00488=114.728,-49.613,26.396,179.9969,-0.0071,0.0000
C00489=113.088,-53.172,26.370,179.9688,-0.0646,0.0000
C00490=111.111,-56.745,26.330,179.8867,-0.1749,0.0000
C00491=108.697,-59.989,26.290,178.9161,-1.2658,0.0000
C00492=106.220,-62.476,26.240,176.8856,-2.5833,0.0000
C00493=104.021,-63.923,26.145,173.9577,-3.0001,0.0000
C00494=101.965,-64.806,25.947,169.9518,-3.7561,0.0000
C00495=99.954,-65.693,25.677,164.7594,-7.3840,0.0000
C00496=97.833,-67.095,25.402,161.1325,-14.3660,0.0000
C00497=95.240,-69.647,25.193,161.0506,-20.6073,0.0000
C00498=91.707,-73.859,25.107,161.1561,-22.3142,0.0000
C00499=87.773,-78.472,25.104,160.3874,-21.7796,0.0000
C00500=83.255,-83.255,25.106,159.2743,-20.7254,0.0000
C00501=78.472,-87.773,25.104,158.2207,-19.6128,0.0000
C00502=73.859,-91.707,25.107,157.6861,-18.8442,0.0000
C00503=69.647,-95.240,25.193,159.3925,-18.9491,0.0000
C00504=67.095,-97.833,25.402,165.6340,-18.8675,0.0000
C00505=65.693,-99.954,25.677,172.6160,-15.2406,0.0000
C00506=64.806,-101.965,25.947,176.2439,-10.0482,0.0000
C00507=63.923,-104.021,26.145,176.9999,-6.0423,0.0000
C00508=62.476,-106.220,26.240,177.4167,-3.1144,0.0000
C00509=59.989,-108.697,26.290,178.7342,-1.0839,0.0000
C00510=56.745,-111.111,26.330,179.8251,-0.1133,0.0000
C00511=53.172,-113.088,26.370,179.9354,-0.0312,0.0000
C00512=49.613,-114.728,26.396,179.9929,-0.0031,0.0000
C00513=46.044,-116.206,26.396,179.9928,-0.0028,0.0000
C00514=42.367,-117.564,26.370,179.9323,-0.0236,0.0000
C00515=38.442,-118.692,26.330,179.7962,-0.0436,0.0000
C00516=34.441,-119.279,26.290,178.3387,-0.1287,0.0000
C00517=30.931,-119.286,26.240,175.9744,0.3765,0.0000
C00518=28.354,-118.754,26.145,173.6147,2.1641,0.0000
C00519=26.275,-117.926,25.947,170.2564,4.5098,0.0000
C00520=24.226,-117.130,25.677,164.1300,5.7683,0.0000
C00521=21.735,-116.622,25.402,157.0835,3.4645,0.0000
C00522=18.097,-116.593,25.193,153.0392,-1.3238,0.0000
C00523=12.620,-117.073,25.107,152.0079,-2.7988,0.0000
C00524=6.577,-117.553,25.104,151.8757,-1.7507,0.0000
C00525=0.000,-117.740,25.106,151.8484,0.0003,0.0000
C00526=0.000,-117.740,25.106,151.8484,0.0003,0.0000
C00527=-6.577,-117.553,25.104,151.8757,1.7504,0.0000
C00528=-12.620,-117.073,25.107,152.0079,2.7983,0.0000
C00529=-18.097,-116.593,25.193,153.0392,1.3242,0.0000
C00530=-21.735,-116.622,25.402,157.0835,-3.4645,0.0000
C00531=-24.226,-117.130,25.677,164.1300,-5.7683,0.0000
C00532=-26.275,-117.926,25.947,170.2564,-4.5098,0.0000
C00533=-28.354,-118.754,26.145,173.6147,-2.1641,0.0000
C00534=-30.931,-119.286,26.240,175.9744,-0.3765,0.0000
C00535=-34.441,-119.279,26.290,178.3387,0.1287,0.0000
C00536=-38.442,-118.692,26.330,179.7962,0.0436,0.0000
C00537=-42.367,-117.564,26.370,179.9323,0.0236,0.0000
C00538=-46.044,-116.206,26.396,179.9928,0.0028,0.0000
C00539=-49.613,-114.728,26.396,179.9929,0.0031,0.0000
C00540=-53.172,-113.088,26.370,179.9354,0.0312,0.0000
C00541=-56.745,-111.111,26.330,179.8251,0.1133,0.0000
C00542=-59.989,-108.697,26.290,178.7342,1.0839,0.0000
C00543=-62.476,-106.220,26.240,177.4167,3.1144,0.0000
C00544=-63.923,-104.021,26.145,176.9999,6.0423,0.0000
C00545=-64.806,-101.965,25.947,176.2439,10.0482,0.0000
C00546=-65.693,-99.954,25.677,172.6160,15.2406,0.0000
C00547=-67.095,-97.833,25.402,165.6340,18.8675,0.0000
C00548=-69.647,-95.240,25.193,159.3927,18.9494,0.0000
C00549=-73.859,-91.707,25.107,157.6858,18.8439,0.0000
C00550=-78.472,-87.773,25.104,158.2204,19.6126,0.0000
C00551=-83.255,-83.255,25.106,159.2746,20.7257,0.0000
C00552=-87.773,-78.472,25.104,160.3872,21.7793,0.0000
C00553=-91.707,-73.859,25.107,161.1558,22.3139,0.0000
C00554=-95.240,-69.647,25.193,161.0509,20.6075,0.0000
C00555=-97.833,-67.095,25.402,161.1325,14.3660,0.0000
C00556=-99.954,-65.693,25.677,164.7594,7.3840,0.0000
C00557=-101.965,-64.806,25.947,169.9518,3.7561,0.0000
C00558=-104.021,-63.923,26.145,173.9577,3.0001,0.0000
C00559=-106.220,-62.476,26.240,176.8856,2.5833,0.0000
C00560=-108.697,-59.989,26.290,178.9161,1.2658,0.0000
C00561=-111.111,-56.745,26.330,179.8867,0.1749,0.0000
C00562=-113.088,-53.172,26.370,179.9688,0.0646,0.0000
C00563=-114.728,-49.613,26.396,179.9969,0.0071,0.0000
C00564=-116.206,-46.044,26.396,179.9972,0.0072,0.0000
C00565=-117.564,-42.367,26.370,179.9764,0.0677,0.0000
C00566=-118.692,-38.442,26.330,179.9564,0.2038,0.0000
C00567=-119.279,-34.441,26.290,179.8713,1.6613,0.0000
C00568=-119.286,-30.931,26.240,-179.6235,4.0256,0.0000
C00569=-118.754,-28.354,26.145,-177.8359,6.3853,0.0000
C00570=-117.926,-26.275,25.947,-175.4902,9.7436,0.0000
C00571=-117.130,-24.226,25.677,-174.2317,15.8700,0.0000
C00572=-116.622,-21.735,25.402,-176.5355,22.9165,0.0000
C00573=-116.593,-18.097,25.193,178.6762,26.9608,0.0000
C00574=-117.073,-12.620,25.107,177.2012,27.9921,0.0000
C00575=-117.553,-6.577,25.104,178.2493,28.1243,0.0000
C00576=-117.740,0.000,25.106,-179.9997,28.1516,0.0000
C00577=-117.553,6.577,25.104,-178.2496,28.1243,0.0000
C00578=-117.073,12.620,25.107,-177.2017,27.9921,0.0000
C00579=-116.593,18.097,25.193,-178.6758,26.9608,0.0000
C00580=-116.622,21.735,25.402,176.5355,22.9165,0.0000
C00581=-117.130,24.226,25.677,174.2317,15.8700,0.0000
C00582=-117.926,26.275,25.947,175.4902,9.7436,0.0000
C00583=-118.754,28.354,26.145,177.8359,6.3853,0.0000
C00584=-119.286,30.931,26.240,179.6235,4.0256,0.0000
C00585=-119.279,34.441,26.290,-179.8713,1.6613,0.0000
C00586=-118.692,38.442,26.330,-179.9564,0.2038,0.0000
C00587=-117.564,42.367,26.370,-179.9764,0.0677,0.0000
C00588=-116.206,46.044,26.396,-179.9972,0.0072,0.0000
C00589=-114.728,49.613,26.396,-179.9969,0.0071,0.0000
C00590=-113.088,53.172,26.370,-179.9688,0.0646,0.0000
C00591=-111.111,56.745,26.330,-179.8867,0.1749,0.0000
C00592=-108.697,59.989,26.290,-178.9161,1.2658,0.0000
C00593=-106.220,62.476,26.240,-176.8856,2.5833,0.0000
C00594=-104.021,63.923,26.145,-173.9577,3.0001,0.0000
C00595=-101.965,64.806,25.947,-169.9518,3.7561,0.0000
C00596=-99.954,65.693,25.677,-164.7594,7.3840,0.0000
C00597=-97.833,67.095,25.402,-161.1325,14.3660,0.0000
C00598=-95.240,69.647,25.193,-161.0506,20.6073,0.0000
C00599=-91.707,73.859,25.107,-161.1561,22.3142,0.0000
C00600=-87.773,78.472,25.104,-160.3874,21.7796,0.0000
C00601=-83.255,83.255,25.106,-159.2743,20.7254,0.0000
C00602=-78.472,87.773,25.104,-158.2207,19.6128,0.0000
C00603=-73.859,91.707,25.107,-157.6861,18.8442,0.0000
C00604=-69.647,95.240,25.193,-159.3925,18.9491,0.0000
C00605=-67.095,97.833,25.402,-165.6340,18.8675,0.0000
C00606=-65.693,99.954,25.677,-172.6160,15.2406,0.0000
C00607=-64.806,101.965,25.947,-176.2439,10.0482,0.0000
C00608=-63.923,104.021,26.145,-176.9999,6.0423,0.0000
C00609=-62.476,106.220,26.240,-177.4167,3.1144,0.0000
C00610=-59.989,108.697,26.290,-178.7342,1.0839,0.0000
C00611=-56.745,111.111,26.330,-179.8251,0.1133,0.0000
C00612=-53.172,113.088,26.370,-179.9354,0.0312,0.0000
C00613=-49.613,114.728,26.396,-179.9929,0.0031,0.0000
C00614=-46.044,116.206,26.396,-179.9928,0.0028,0.0000
C00615=-42.367,117.564,26.370,-179.9323,0.0236,0.0000
C00616=-38.442,118.692,26.330,-179.7962,0.0436,0.0000
C00617=-34.441,119.279,26.290,-178.3387,0.1287,0.0000
C00618=-30.931,119.286,26.240,-175.9744,-0.3765,0.0000
C00619=-28.354,118.754,26.145,-173.6147,-2.1641,0.0000
C00620=-26.275,117.926,25.947,-170.2564,-4.5098,0.0000
C00621=-24.226,117.130,25.677,-164.1300,-5.7683,0.0000
C00622=-21.735,116.622,25.402,-157.0835,-3.4645,0.0000
C00623=-18.097,116.593,25.193,-153.0392,1.3242,0.0000
C00624=-12.620,117.073,25.107,-152.0079,2.7983,0.0000
C00625=-6.577,117.553,25.104,-151.8757,1.7504,0.0000
C00626=0.000,117.740,25.106,-151.8484,0.0003,0.0000
C00627=0.000,116.679,27.034,-150.5252,0.0003,0.0000
C00628=6.480,116.496,27.031,-150.5533,-1.8438,0.0000
C00629=12.457,116.025,27.035,-150.6875,-2.8625,0.0000
C00630=17.898,115.583,27.137,-151.8014,-0.8610,0.0000
C00631=21.492,115.706,27.387,-156.6336,4.8857,0.0000
C00632=23.949,116.359,27.719,-164.8085,6.9131,0.0000
C00633=25.975,117.338,28.046,-171.2616,5.0049,0.0000
C00634=28.031,118.371,28.287,-174.3842,2.4458,0.0000
C00635=30.581,119.095,28.404,-176.3475,0.5561,0.0000
C00636=34.111,119.239,28.464,-178.5229,-0.0669,0.0000
C00637=38.181,118.740,28.514,-179.8949,-0.0207,0.0000
C00638=42.202,117.618,28.563,-179.9393,-0.0210,0.0000
C00639=45.987,116.228,28.596,-179.9937,-0.0025,0.0000
C00640=49.668,114.704,28.596,-179.9938,-0.0027,0.0000
C00641=53.328,113.010,28.563,-179.9423,-0.0281,0.0000
C00642=56.964,110.960,28.514,-179.9110,-0.0596,0.0000
C00643=60.195,108.435,28.464,-178.9082,-0.9973,0.0000
C00644=62.589,105.837,28.404,-177.8081,-2.9768,0.0000
C00645=63.879,103.522,28.287,-177.7480,-5.6954,0.0000
C00646=64.604,101.338,28.046,-177.3227,-9.6822,0.0000
C00647=65.344,99.213,27.719,-173.9340,-15.5220,0.0000
C00648=66.619,97.014,27.387,-166.2306,-20.0997,0.0000
C00649=69.074,94.385,27.137,-158.7065,-20.2288,0.0000
C00650=73.234,90.850,27.035,-156.6178,-19.8828,0.0000
C00651=77.793,86.957,27.031,-157.1223,-20.6279,0.0000
C00652=82.505,82.505,27.034,-158.2160,-21.7844,0.0000
C00653=86.957,77.793,27.031,-159.3719,-22.8774,0.0000
C00654=90.851,73.234,27.035,-160.1168,-23.3818,0.0000
C00655=94.385,69.074,27.137,-159.7715,-21.2937,0.0000
C00656=97.014,66.619,27.387,-159.9003,-13.7694,0.0000
C00657=99.213,65.344,27.719,-164.4780,-6.0660,0.0000
C00658=101.338,64.604,28.046,-170.3178,-2.6773,0.0000
C00659=103.522,63.879,28.287,-174.3046,-2.2520,0.0000
C00660=105.837,62.589,28.404,-177.0232,-2.1919,0.0000
C00661=108.435,60.195,28.464,-179.0027,-1.0918,0.0000
C00662=110.960,56.964,28.514,-179.9404,-0.0890,0.0000
C00663=113.010,53.328,28.563,-179.9719,-0.0577,0.0000
C00664=114.704,49.668,28.596,-179.9973,-0.0062,0.0000
C00665=116.228,45.987,28.596,-179.9975,-0.0063,0.0000
C00666=117.618,42.202,28.563,-179.9790,-0.0607,0.0000
C00667=118.740,38.181,28.514,-179.9793,-0.1051,0.0000
C00668=119.239,34.111,28.464,-179.9331,-1.4771,0.0000
C00669=119.095,30.581,28.404,179.4439,-3.6525,0.0000
C00670=118.371,28.031,28.287,177.5542,-5.6158,0.0000
C00671=117.338,25.975,28.046,174.9951,-8.7384,0.0000
C00672=116.359,23.949,27.719,173.0869,-15.1915,0.0000
C00673=115.706,21.492,27.387,175.1143,-23.3664,0.0000
C00674=115.583,17.898,27.137,-179.1390,-28.1986,0.0000
C00675=116.025,12.457,27.035,-177.1375,-29.3125,0.0000
C00676=116.496,6.480,27.031,-178.1562,-29.4467,0.0000
C00677=116.679,0.000,27.034,179.9997,-29.4748,0.0000
C00678=116.496,-6.480,27.031,178.1566,-29.4467,0.0000
C00679=116.025,-12.457,27.035,177.1381,-29.3125,0.0000
C00680=115.583,-17.898,27.137,179.1386,-28.1986,0.0000
C00681=115.706,-21.492,27.387,-175.1143,-23.3664,0.0000
C00682=116.359,-23.949,27.719,-173.0869,-15.1915,0.0000
C00683=117.338,-25.975,28.046,-174.9951,-8.7384,0.0000
C00684=118.371,-28.031,28.287,-177.5542,-5.6158,0.0000
C00685=119.095,-30.581,28.404,-179.4439,-3.6525,0.0000
C00686=119.239,-34.111,28.464,179.9331,-1.4771,0.0000
C00687=118.740,-38.181,28.514,179.9793,-0.1051,0.0000
C00688=117.618,-42.202,28.563,179.9790,-0.0607,0.0000
C00689=116.228,-45.987,28.596,179.9975,-0.0063,0.0000
C00690=114.704,-49.668,28.596,179.9973,-0.0062,0.0000
C00691=113.010,-53.328,28.563,179.9719,-0.0577,0.0000
C00692=110.960,-56.964,28.514,179.9404,-0.0890,0.0000
C00693=108.435,-60.195,28.464,179.0027,-1.0918,0.0000
C00694=105.837,-62.589,28.404,177.0232,-2.1919,0.0000
C00695=103.522,-63.879,28.287,174.3046,-2.2520,0.0000
C00696=101.338,-64.604,28.046,170.3178,-2.6773,0.0000
C00697=99.213,-65.344,27.719,164.4780,-6.0660,0.0000
C00698=97.014,-66.619,27.387,159.9003,-13.7694,0.0000
C00699=94.385,-69.074,27.137,159.7712,-21.2935,0.0000
C00700=90.850,-73.234,27.035,160.1172,-23.3822,0.0000
C00701=86.957,-77.793,27.031,159.3721,-22.8777,0.0000
C00702=82.505,-82.505,27.034,158.2156,-21.7840,0.0000
C00703=77.793,-86.957,27.031,157.1226,-20.6281,0.0000
C00704=73.234,-90.851,27.035,156.6182,-19.8832,0.0000
C00705=69.074,-94.385,27.137,158.7063,-20.2285,0.0000
C00706=66.619,-97.014,27.387,166.2306,-20.0997,0.0000
C00707=65.344,-99.213,27.719,173.9340,-15.5220,0.0000
C00708=64.604,-101.338,28.046,177.3227,-9.6822,0.0000
C00709=63.879,-103.522,28.287,177.7480,-5.6954,0.0000
C00710=62.589,-105.837,28.404,177.8081,-2.9768,0.0000
C00711=60.195,-108.435,28.464,178.9082,-0.9973,0.0000
C00712=56.964,-110.960,28.514,179.9110,-0.0596,0.0000
C00713=53.328,-113.010,28.563,179.9423,-0.0281,0.0000
C00714=49.668,-114.704,28.596,179.9938,-0.0027,0.0000
C00715=45.987,-116.228,28.596,179.9937,-0.0025,0.0000
C00716=42.202,-117.618,28.563,179.9393,-0.0210,0.0000
C00717=38.181,-118.740,28.514,179.8949,-0.0207,0.0000
C00718=34.111,-119.239,28.464,178.5229,-0.0669,0.0000
C00719=30.581,-119.095,28.404,176.3475,0.5561,0.0000
C00720=28.031,-118.371,28.287,174.3842,2.4458,0.0000
C00721=25.975,-117.338,28.046,171.2616,5.0049,0.0000
C00722=23.949,-116.359,27.719,164.8085,6.9131,0.0000
C00723=21.492,-115.706,27.387,156.6336,4.8857,0.0000
C00724=17.898,-115.583,27.137,151.8014,-0.8610,0.0000
C00725=12.457,-116.025,27.035,150.6875,-2.8625,0.0000
C00726=6.480,-116.496,27.031,150.5533,-1.8438,0.0000
C00727=0.000,-116.679,27.034,150.5252,0.0003,0.0000
C00728=0.000,-116.679,27.034,150.5252,0.0003,0.0000
C00729=-6.480,-116.496,27.031,150.5533,1.8434,0.0000
C00730=-12.457,-116.025,27.035,150.6875,2.8619,0.0000
C00731=-17.898,-115.583,27.137,151.8014,0.8614,0.0000
C00732=-21.492,-115.706,27.387,156.6336,-4.8857,0.0000
C00733=-23.949,-116.359,27.719,164.8085,-6.9131,0.0000
C00734=-25.975,-117.338,28.046,171.2616,-5.0049,0.0000
C00735=-28.031,-118.371,28.287,174.3842,-2.4458,0.0000
C00736=-30.581,-119.095,28.404,176.3475,-0.5561,0.0000
C00737=-34.111,-119.239,28.464,178.5229,0.0669,0.0000
C00738=-38.181,-118.740,28.514,179.8949,0.0207,0.0000
C00739=-42.202,-117.618,28.563,179.9393,0.0210,0.0000
C00740=-45.987,-116.228,28.596,179.9937,0.0025,0.0000
C00741=-49.668,-114.704,28.596,179.9938,0.0027,0.0000
C00742=-53.328,-113.010,28.563,179.9423,0.0281,0.0000
C00743=-56.964,-110.960,28.514,179.9110,0.0596,0.0000
C00744=-60.195,-108.435,28.464,178.9082,0.9973,0.0000
C00745=-62.589,-105.837,28.404,177.8081,2.9768,0.0000
C00746=-63.879,-103.522,28.287,177.7480,5.6954,0.0000
C00747=-64.604,-101.338,28.046,177.3227,9.6822,0.0000
C00748=-65.344,-99.213,27.719,173.9340,15.5220,0.0000
C00749=-66.619,-97.014,27.387,166.2306,20.0997,0.0000
C00750=-69.074,-94.385,27.137,158.7065,20.2288,0.0000
C00751=-73.234,-90.850,27.035,156.6178,19.8828,0.0000
C00752=-77.793,-86.957,27.031,157.1223,20.6279,0.0000
C00753=-82.505,-82.505,27.034,158.2160,21.7844,0.0000
C00754=-86.957,-77.793,27.031,159.3719,22.8774,0.0000
C00755=-90.851,-73.234,27.035,160.1168,23.3818,0.0000
C00756=-94.385,-69.074,27.137,159.7715,21.2937,0.0000
C00757=-97.014,-66.619,27.387,159.9003,13.7694,0.0000
C00758=-99.213,-65.344,27.719,164.4780,6.0660,0.0000
C00759=-101.338,-64.604,28.046,170.3178,2.6773,0.0000
C00760=-103.522,-63.879,28.287,174.3046,2.2520,0.0000
C00761=-105.837,-62.589,28.404,177.0232,2.1919,0.0000
C00762=-108.435,-60.195,28.464,179.0027,1.0918,0.0000
C00763=-110.960,-56.964,28.514,179.9404,0.0890,0.0000
C00764=-113.010,-53.328,28.563,179.9719,0.0577,0.0000
C00765=-114.704,-49.668,28.596,179.9973,0.0062,0.0000
C00766=-116.228,-45.987,28.596,179.9975,0.0063,0.0000
C00767=-117.618,-42.202,28.563,179.9790,0.0607,0.0000
C00768=-118.740,-38.181,28.514,179.9793,0.1051,0.0000
C00769=-119.239,-34.111,28.464,179.9331,1.4771,0.0000
C00770=-119.095,-30.581,28.404,-179.4439,3.6525,0.0000
C00771=-118.371,-28.031,28.287,-177.5542,5.6158,0.0000
C00772=-117.338,-25.975,28.046,-174.9951,8.7384,0.0000
C00773=-116.359,-23.949,27.719,-173.0869,15.1915,0.0000
C00774=-115.706,-21.492,27.387,-175.1143,23.3664,0.0000
C00775=-115.583,-17.898,27.137,179.1390,28.1986,0.0000
C00776=-116.025,-12.457,27.035,177.1375,29.3125,0.0000
C00777=-116.496,-6.480,27.031,178.1562,29.4467,0.0000
C00778=-116.679,0.000,27.034,-179.9997,29.4748,0.0000
C00779=-116.496,6.480,27.031,-178.1566,29.4467,0.0000
C00780=-116.025,12.457,27.035,-177.1381,29.3125,0.0000
C00781=-115.583,17.898,27.137,-179.1386,28.1986,0.0000
C00782=-115.706,21.492,27.387,175.1143,23.3664,0.0000
C00783=-116.359,23.949,27.719,173.0869,15.1915,0.0000
C00784=-117.338,25.975,28.046,174.9951,8.7384,0.0000
C00785=-118.371,28.031,28.287,177.5542,5.6158,0.0000
C00786=-119.095,30.581,28.404,179.4439,3.6525,0.0000
C00787=-119.239,34.111,28.464,-179.9331,1.4771,0.0000
C00788=-118.740,38.181,28.514,-179.9793,0.1051,0.0000
C00789=-117.618,42.202,28.563,-179.9790,0.0607,0.0000
C00790=-116.228,45.987,28.596,-179.9975,0.0063,0.0000
C00791=-114.704,49.668,28.596,-179.9973,0.0062,0.0000
C00792=-113.010,53.328,28.563,-179.9719,0.0577,0.0000
C00793=-110.960,56.964,28.514,-179.9404,0.0890,0.0000
C00794=-108.435,60.195,28.464,-179.0027,1.0918,0.0000
C00795=-105.837,62.589,28.404,-177.0232,2.1919,0.0000
C00796=-103.522,63.879,28.287,-174.3046,2.2520,0.0000
C00797=-101.338,64.604,28.046,-170.3178,2.6773,0.0000
C00798=-99.213,65.344,27.719,-164.4780,6.0660,0.0000
C00799=-97.014,66.619,27.387,-159.9003,13.7694,0.0000
C00800=-94.385,69.074,27.137,-159.7712,21.2935,0.0000
C00801=-90.850,73.234,27.035,-160.1172,23.3822,0.0000
C00802=-86.957,77.793,27.031,-159.3721,22.8777,0.0000
C00803=-82.505,82.505,27.034,-158.2156,21.7840,0.0000
C00804=-77.793,86.957,27.031,-157.1226,20.6281,0.0000
C00805=-73.234,90.851,27.035,-156.6182,19.8832,0.0000
C00806=-69.074,94.385,27.137,-158.7063,20.2285,0.0000
C00807=-66.619,97.014,27.387,-166.2306,20.0997,0.0000
C00808=-65.344,99.213,27.719,-173.9340,15.5220,0.0000
C00809=-64.604,101.338,28.046,-177.3227,9.6822,0.0000
C00810=-63.879,103.522,28.287,-177.7480,5.6954,0.0000
C00811=-62.589,105.837,28.404,-177.8081,2.9768,0.0000
C00812=-60.195,108.435,28.464,-178.9082,0.9973,0.0000
C00813=-56.964,110.960,28.514,-179.9110,0.0596,0.0000
C00814=-53.328,113.010,28.563,-179.9423,0.0281,0.0000
C00815=-49.668,114.704,28.596,-179.9938,0.0027,0.0000
C00816=-45.987,116.228,28.596,-179.9937,0.0025,0.0000
C00817=-42.202,117.618,28.563,-179.9393,0.0210,0.0000
C00818=-38.181,118.740,28.514,-179.8949,0.0207,0.0000
C00819=-34.111,119.239,28.464,-178.5229,0.0669,0.0000
C00820=-30.581,119.095,28.404,-176.3475,-0.5561,0.0000
C00821=-28.031,118.371,28.287,-174.3842,-2.4458,0.0000
C00822=-25.975,117.338,28.046,-171.2616,-5.0049,0.0000
C00823=-23.949,116.359,27.719,-164.8085,-6.9131,0.0000
C00824=-21.492,115.706,27.387,-156.6336,-4.8857,0.0000
C00825=-17.898,115.583,27.137,-151.8014,0.8614,0.0000
C00826=-12.457,116.025,27.035,-150.6875,2.8619,0.0000
C00827=-6.480,116.496,27.031,-150.5533,1.8434,0.0000
C00828=0.000,116.679,27.034,-150.5252,0.0003,0.0000
C00829=0.000,115.576,28.937,-149.3196,0.0003,0.0000
C00830=6.379,115.397,28.934,-149.3483,-1.9296,0.0000
C00831=12.287,114.936,28.939,-149.4843,-2.9007,0.0000
C00832=17.690,114.532,29.058,-150.6979,-0.3111,0.0000
C00833=21.239,114.751,29.353,-156.4871,6.3635,0.0000
C00834=23.659,115.553,29.745,-165.7977,7.8311,0.0000
C00835=25.660,116.723,30.134,-172.4231,5.2207,0.0000
C00836=27.693,117.967,30.423,-175.2991,2.5322,0.0000
C00837=30.212,118.894,30.563,-176.8393,0.6777,0.0000
C00838=33.764,119.197,30.636,-178.7547,-0.0152,0.0000
C00839=37.905,118.790,30.696,179.9918,0.0015,0.0000
C00840=42.028,117.676,30.755,-179.9477,-0.0179,0.0000
C00841=45.928,116.251,30.795,-179.9948,-0.0020,0.0000
C00842=49.726,114.678,30.795,-179.9948,-0.0023,0.0000
C00843=53.491,112.927,30.755,-179.9504,-0.0243,0.0000
C00844=57.194,110.800,30.696,179.9931,0.0048,0.0000
C00845=60.411,108.160,30.636,-179.1086,-0.8698,0.0000
C00846=62.708,105.434,30.563,-178.2426,-2.7145,0.0000
C00847=63.834,102.997,30.423,-178.4606,-5.1096,0.0000
C00848=64.391,100.680,30.134,-178.3132,-9.0158,0.0000
C00849=64.979,98.438,29.745,-175.3291,-15.4406,0.0000
C00850=66.123,96.159,29.353,-167.1131,-21.1318,0.0000
C00851=68.477,93.495,29.058,-158.1649,-21.4551,0.0000
C00852=72.583,89.960,28.939,-155.6481,-20.8543,0.0000
C00853=77.087,86.109,28.934,-156.1131,-21.5650,0.0000
C00854=81.725,81.725,28.937,-157.2410,-22.7594,0.0000
C00855=86.109,77.088,28.934,-158.4348,-23.8867,0.0000
C00856=89.960,72.583,28.939,-159.1453,-24.3515,0.0000
C00857=93.495,68.477,29.058,-158.5452,-21.8354,0.0000
C00858=96.159,66.123,29.353,-158.8682,-12.8869,0.0000
C00859=98.438,64.979,29.745,-164.5594,-4.6709,0.0000
C00860=100.680,64.391,30.134,-170.9842,-1.6868,0.0000
C00861=102.997,63.834,30.423,-174.8904,-1.5394,0.0000
C00862=105.434,62.708,30.563,-177.2855,-1.7574,0.0000
C00863=108.160,60.411,30.636,-179.1302,-0.8914,0.0000
C00864=110.800,57.194,30.696,179.9952,0.0069,0.0000
C00865=112.927,53.491,30.755,-179.9757,-0.0496,0.0000
C00866=114.678,49.726,30.795,-179.9977,-0.0052,0.0000
C00867=116.251,45.928,30.795,-179.9980,-0.0052,0.0000
C00868=117.676,42.028,30.755,-179.9821,-0.0523,0.0000
C00869=118.790,37.905,30.696,179.9985,0.0082,0.0000
C00870=119.197,33.764,30.636,-179.9848,-1.2453,0.0000
C00871=118.894,30.212,30.563,179.3223,-3.1607,0.0000
C00872=117.967,27.693,30.423,177.4678,-4.7009,0.0000
C00873=116.723,25.660,30.134,174.7793,-7.5769,0.0000
C00874=115.553,23.659,29.745,172.1689,-14.2023,0.0000
C00875=114.751,21.239,29.353,173.6365,-23.5129,0.0000
C00876=114.532,17.690,29.058,-179.6889,-29.3021,0.0000
C00877=114.936,12.287,28.939,-177.0993,-30.5157,0.0000
C00878=115.397,6.379,28.934,-178.0704,-30.6517,0.0000
C00879=115.576,0.000,28.937,179.9997,-30.6804,0.0000
C00880=115.397,-6.379,28.934,178.0709,-30.6517,0.0000
C00881=114.936,-12.287,28.939,177.1000,-30.5157,0.0000
C00882=114.532,-17.690,29.058,179.6885,-29.3021,0.0000
C00883=114.751,-21.239,29.353,-173.6365,-23.5129,0.0000
C00884=115.553,-23.659,29.745,-172.1689,-14.2023,0.0000
C00885=116.723,-25.660,30.134,-174.7793,-7.5769,0.0000
C00886=117.967,-27.693,30.423,-177.4678,-4.7009,0.0000
C00887=118.894,-30.212,30.563,-179.3223,-3.1607,0.0000
C00888=119.197,-33.764,30.636,179.9848,-1.2453,0.0000
C00889=118.790,-37.905,30.696,-179.9985,0.0082,0.0000
C00890=117.676,-42.028,30.755,179.9821,-0.0523,0.0000
C00891=116.251,-45.928,30.795,179.9980,-0.0052,0.0000
C00892=114.678,-49.726,30.795,179.9977,-0.0052,0.0000
C00893=112.927,-53.491,30.755,179.9757,-0.0496,0.0000
C00894=110.800,-57.194,30.696,-179.9952,0.0069,0.0000
C00895=108.160,-60.411,30.636,179.1302,-0.8914,0.0000
C00896=105.434,-62.708,30.563,177.2855,-1.7574,0.0000
C00897=102.997,-63.834,30.423,174.8904,-1.5394,0.0000
C00898=100.680,-64.391,30.134,170.9842,-1.6868,0.0000
C00899=98.438,-64.979,29.745,164.5594,-4.6709,0.0000
C00900=96.159,-66.123,29.353,158.8682,-12.8869,0.0000
C00901=93.495,-68.477,29.058,158.5449,-21.8351,0.0000
C00902=89.960,-72.583,28.939,159.1457,-24.3519,0.0000
C00903=86.109,-77.087,28.934,158.4350,-23.8869,0.0000
C00904=81.725,-81.725,28.937,157.2406,-22.7590,0.0000
C00905=77.088,-86.109,28.934,156.1133,-21.5652,0.0000
C00906=72.583,-89.960,28.939,155.6485,-20.8547,0.0000
C00907=68.477,-93.495,29.058,158.1646,-21.4548,0.0000
C00908=66.123,-96.159,29.353,167.1131,-21.1318,0.0000
C00909=64.979,-98.438,29.745,175.3291,-15.4406,0.0000
C00910=64.391,-100.680,30.134,178.3132,-9.0158,0.0000
C00911=63.834,-102.997,30.423,178.4606,-5.1096,0.0000
C00912=62.708,-105.434,30.563,178.2426,-2.7145,0.0000
C00913=60.411,-108.160,30.636,179.1086,-0.8698,0.0000
C00914=57.194,-110.800,30.696,-179.9931,0.0048,0.0000
C00915=53.491,-112.927,30.755,179.9504,-0.0243,0.0000
C00916=49.726,-114.678,30.795,179.9948,-0.0023,0.0000
C00917=45.928,-116.251,30.795,179.9948,-0.0020,0.0000
C00918=42.028,-117.676,30.755,179.9477,-0.0179,0.0000
C00919=37.905,-118.790,30.696,-179.9918,0.0015,0.0000
C00920=33.764,-119.197,30.636,178.7547,-0.0152,0.0000
C00921=30.212,-118.894,30.563,176.8393,0.6777,0.0000
C00922=27.693,-117.967,30.423,175.2991,2.5322,0.0000
C00923=25.660,-116.723,30.134,172.4231,5.2207,0.0000
C00924=23.659,-115.553,29.745,165.7977,7.8311,0.0000
C00925=21.239,-114.751,29.353,156.4871,6.3635,0.0000
C00926=17.690,-114.532,29.058,150.6979,-0.3111,0.0000
C00927=12.287,-114.936,28.939,149.4843,-2.9007,0.0000
C00928=6.379,-115.397,28.934,149.3483,-1.9296,0.0000
C00929=0.000,-115.576,28.937,149.3196,0.0003,0.0000
C00930=0.000,-115.576,28.937,149.3196,0.0003,0.0000
C00931=-6.379,-115.397,28.934,149.3483,1.9291,0.0000
C00932=-12.287,-114.936,28.939,149.4843,2.9000,0.0000
C00933=-17.690,-114.532,29.058,150.6979,0.3115,0.0000
C00934=-21.239,-114.751,29.353,156.4871,-6.3635,0.0000
C00935=-23.659,-115.553,29.745,165.7977,-7.8311,0.0000
C00936=-25.660,-116.723,30.134,172.4231,-5.2207,0.0000
C00937=-27.693,-117.967,30.423,175.2991,-2.5322,0.0000
C00938=-30.212,-118.894,30.563,176.8393,-0.6777,0.0000
C00939=-33.764,-119.197,30.636,178.7547,0.0152,0.0000
C00940=-37.905,-118.790,30.696,-179.9918,-0.0015,0.0000
C00941=-42.028,-117.676,30.755,179.9477,0.0179,0.0000
C00942=-45.928,-116.251,30.795,179.9948,0.0020,0.0000
C00943=-49.726,-114.678,30.795,179.9948,0.0023,0.0000
C00944=-53.491,-112.927,30.755,179.9504,0.0243,0.0000
C00945=-57.194,-110.800,30.696,-179.9931,-0.0048,0.0000
C00946=-60.411,-108.160,30.636,179.1086,0.8698,0.0000
C00947=-62.708,-105.434,30.563,178.2426,2.7145,0.0000
C00948=-63.834,-102.997,30.423,178.4606,5.1096,0.0000
C00949=-64.391,-100.680,30.134,178.3132,9.0158,0.0000
C00950=-64.979,-98.438,29.745,175.3291,15.4406,0.0000
C00951=-66.123,-96.159,29.353,167.1131,21.1318,0.0000
C00952=-68.477,-93.495,29.058,158.1649,21.4551,0.0000
C00953=-72.583,-89.960,28.939,155.6481,20.8543,0.0000
C00954=-77.087,-86.109,28.934,156.1131,21.5650,0.0000
C00955=-81.725,-81.725,28.937,157.2410,22.7594,0.0000
C00956=-86.109,-77.088,28.934,158.4348,23.8867,0.0000
C00957=-89.960,-72.583,28.939,159.1453,24.3515,0.0000
C00958=-93.495,-68.477,29.058,158.5452,21.8354,0.0000
C00959=-96.159,-66.123,29.353,158.8682,12.8869,0.0000
C00960=-98.438,-64.979,29.745,164.5594,4.6709,0.0000
C00961=-100.680,-64.391,30.134,170.9842,1.6868,0.0000
C00962=-102.997,-63.834,30.423,174.8904,1.5394,0.0000
C00963=-105.434,-62.708,30.563,177.2855,1.7574,0.0000
C00964=-108.160,-60.411,30.636,179.1302,0.8914,0.0000
C00965=-110.800,-57.194,30.696,-179.9952,-0.0069,0.0000
C00966=-112.927,-53.491,30.755,179.9757,0.0496,0.0000
C00967=-114.678,-49.726,30.795,179.9977,0.0052,0.0000
C00968=-116.251,-45.928,30.795,179.9980,0.0052,0.0000
C00969=-117.676,-42.028,30.755,179.9821,0.0523,0.0000
C00970=-118.790,-37.905,30.696,-179.9985,-0.0082,0.0000
C00971=-119.197,-33.764,30.636,179.9848,1.2453,0.0000
C00972=-118.894,-30.212,30.563,-179.3223,3.1607,0.0000
C00973=-117.967,-27.693,30.423,-177.4678,4.7009,0.0000
C00974=-116.723,-25.660,30.134,-174.7793,7.5769,0.0000
C00975=-115.553,-23.659,29.745,-172.1689,14.2023,0.0000
C00976=-114.751,-21.239,29.353,-173.6365,23.5129,0.0000
C00977=-114.532,-17.690,29.058,179.6889,29.3021,0.0000
C00978=-114.936,-12.287,28.939,177.0993,30.5157,0.0000
C00979=-115.397,-6.379,28.934,178.0704,30.6517,0.0000
C00980=-115.576,0.000,28.937,-179.9997,30.6804,0.0000
C00981=-115.397,6.379,28.934,-178.0709,30.6517,0.0000
C00982=-114.936,12.287,28.939,-177.1000,30.5157,0.0000
C00983=-114.532,17.690,29.058,-179.6885,29.3021,0.0000
C00984=-114.751,21.239,29.353,173.6365,23.5129,0.0000
C00985=-115.553,23.659,29.745,172.1689,14.2023,0.0000
C00986=-116.723,25.660,30.134,174.7793,7.5769,0.0000
C00987=-117.967,27.693,30.423,177.4678,4.7009,0.0000
C00988=-118.894,30.212,30.563,179.3223,3.1607,0.0000
C00989=-119.197,33.764,30.636,-179.9848,1.2453,0.0000
C00990=-118.790,37.905,30.696,179.9985,-0.0082,0.0000
C00991=-117.676,42.028,30.755,-179.9821,0.0523,0.0000
C00992=-116.251,45.928,30.795,-179.9980,0.0052,0.0000
C00993=-114.678,49.726,30.795,-179.9977,0.0052,0.0000
C00994=-112.927,53.491,30.755,-179.9757,0.0496,0.0000
C00995=-110.800,57.194,30.696,179.9952,-0.0069,0.0000
C00996=-108.160,60.411,30.636,-179.1302,0.8914,0.0000
C00997=-105.434,62.708,30.563,-177.2855,1.7574,0.0000
C00998=-102.997,63.834,30.423,-174.8904,1.5394,0.0000
C00999=-100.680,64.391,30.134,-170.9842,1.6868,0.0000
C01000=-98.438,64.979,29.745,-164.5594,4.6709,0.0000
C01001=-96.159,66.123,29.353,-158.8682,12.8869,0.0000
C01002=-93.495,68.477,29.058,-158.5449,21.8351,0.0000
C01003=-89.960,72.583,28.939,-159.1457,24.3519,0.0000
C01004=-86.109,77.087,28.934,-158.4350,23.8869,0.0000
C01005=-81.725,81.725,28.937,-157.2406,22.7590,0.0000
C01006=-77.088,86.109,28.934,-156.1133,21.5652,0.0000
C01007=-72.583,89.960,28.939,-155.6485,20.8547,0.0000
C01008=-68.477,93.495,29.058,-158.1646,21.4548,0.0000
C01009=-66.123,96.159,29.353,-167.1131,21.1318,0.0000
C01010=-64.979,98.438,29.745,-175.3291,15.4406,0.0000
C01011=-64.391,100.680,30.134,-178.3132,9.0158,0.0000
C01012=-63.834,102.997,30.423,-178.4606,5.1096,0.0000
C01013=-62.708,105.434,30.563,-178.2426,2.7145,0.0000
C01014=-60.411,108.160,30.636,-179.1086,0.8698,0.0000
C01015=-57.194,110.800,30.696,179.9931,-0.0048,0.0000
C01016=-53.491,112.927,30.755,-179.9504,0.0243,0.0000
C01017=-49.726,114.678,30.795,-179.9948,0.0023,0.0000
C01018=-45.928,116.251,30.795,-179.9948,0.0020,0.0000
C01019=-42.028,117.676,30.755,-179.9477,0.0179,0.0000
C01020=-37.905,118.790,30.696,179.9918,-0.0015,0.0000
C01021=-33.764,119.197,30.636,-178.7547,0.0152,0.0000
C01022=-30.212,118.894,30.563,-176.8393,-0.6777,0.0000
C01023=-27.693,117.967,30.423,-175.2991,-2.5322,0.0000
C01024=-25.660,116.723,30.134,-172.4231,-5.2207,0.0000
C01025=-23.659,115.553,29.745,-165.7977,-7.8311,0.0000
C01026=-21.239,114.751,29.353,-156.4871,-6.3635,0.0000
C01027=-17.690,114.532,29.058,-150.6979,0.3115,0.0000
C01028=-12.287,114.936,28.939,-149.4843,2.9000,0.0000
C01029=-6.379,115.397,28.934,-149.3483,1.9291,0.0000
C01030=0.000,115.576,28.937,-149.3196,0.0003,0.0000
C01031=0.000,114.436,30.818,-148.2225,0.0004,0.0000
C01032=6.275,114.260,30.814,-148.2518,-2.0082,0.0000
C01033=12.112,113.809,30.820,-148.3894,-2.9141,0.0000
C01034=17.476,113.444,30.958,-149.7238,0.3209,0.0000
C01035=20.976,113.761,31.300,-156.6467,7.8338,0.0000
C01036=23.358,114.715,31.757,-167.0185,8.4695,0.0000
C01037=25.331,116.081,32.213,-173.6439,5.1590,0.0000
C01038=27.339,117.546,32.553,-176.2883,2.4064,0.0000
C01039=29.826,118.684,32.719,-177.4308,0.7190,0.0000
C01040=33.400,119.154,32.806,-179.0289,0.0208,0.0000
C01041=37.617,118.843,32.876,179.8658,0.0220,0.0000
C01042=41.845,117.736,32.947,-179.9573,-0.0145,0.0000
C01043=45.866,116.275,32.994,-179.9960,-0.0016,0.0000
C01044=49.786,114.651,32.994,-179.9960,-0.0018,0.0000
C01045=53.663,112.841,32.947,-179.9596,-0.0199,0.0000
C01046=57.435,110.633,32.876,179.8895,0.0793,0.0000
C01047=60.637,107.872,32.806,-179.3280,-0.7014,0.0000
C01048=62.832,105.013,32.719,-178.6908,-2.3251,0.0000
C01049=63.786,102.449,32.553,-179.0744,-4.3226,0.0000
C01050=64.170,99.994,32.213,-179.1450,-8.1161,0.0000
C01051=64.599,97.632,31.757,-176.6969,-15.0188,0.0000
C01052=65.609,95.273,31.300,-168.2488,-21.9295,0.0000
C01053=67.860,92.574,30.958,-157.7631,-22.6247,0.0000
C01054=71.911,89.039,30.820,-154.7706,-21.7619,0.0000
C01055=76.357,85.231,30.814,-155.1873,-22.4282,0.0000
C01056=80.918,80.918,30.818,-156.3449,-23.6556,0.0000
C01057=85.231,76.357,30.814,-157.5715,-24.8125,0.0000
C01058=89.040,71.910,30.820,-158.2376,-25.2289,0.0000
C01059=92.574,67.860,30.958,-157.3756,-22.2373,0.0000
C01060=95.273,65.609,31.300,-158.0705,-11.7512,0.0000
C01061=97.632,64.599,31.757,-164.9812,-3.3031,0.0000
C01062=99.994,64.170,32.213,-171.8839,-0.8550,0.0000
C01063=102.449,63.786,32.553,-175.6774,-0.9256,0.0000
C01064=105.013,62.832,32.719,-177.6749,-1.3092,0.0000
C01065=107.872,60.637,32.806,-179.2986,-0.6720,0.0000
C01066=110.633,57.435,32.876,179.9207,0.1105,0.0000
C01067=112.841,53.663,32.947,-179.9801,-0.0404,0.0000
C01068=114.651,49.786,32.994,-179.9982,-0.0040,0.0000
C01069=116.275,45.866,32.994,-179.9984,-0.0040,0.0000
C01070=117.736,41.845,32.947,-179.9855,-0.0427,0.0000
C01071=118.843,37.617,32.876,179.9780,0.1342,0.0000
C01072=119.154,33.400,32.806,179.9792,-0.9711,0.0000
C01073=118.684,29.826,32.719,179.2810,-2.5692,0.0000
C01074=117.546,27.339,32.553,177.5936,-3.7117,0.0000
C01075=116.081,25.331,32.213,174.8410,-6.3561,0.0000
C01076=114.715,23.358,31.757,171.5305,-12.9815,0.0000
C01077=113.761,20.976,31.300,172.1662,-23.3533,0.0000
C01078=113.444,17.476,30.958,179.6791,-30.2762,0.0000
C01079=113.809,12.112,30.820,-177.0859,-31.6106,0.0000
C01080=114.260,6.275,30.814,-177.9918,-31.7482,0.0000
C01081=114.436,0.000,30.818,179.9996,-31.7775,0.0000
C01082=114.260,-6.275,30.814,177.9923,-31.7482,0.0000
C01083=113.809,-12.112,30.820,177.0867,-31.6106,0.0000
C01084=113.444,-17.476,30.958,-179.6796,-30.2762,0.0000
C01085=113.761,-20.976,31.300,-172.1662,-23.3533,0.0000
C01086=114.715,-23.358,31.757,-171.5305,-12.9815,0.0000
C01087=116.081,-25.331,32.213,-174.8410,-6.3561,0.0000
C01088=117.546,-27.339,32.553,-177.5936,-3.7117,0.0000
C01089=118.684,-29.826,32.719,-179.2810,-2.5692,0.0000
C01090=119.154,-33.400,32.806,-179.9792,-0.9711,0.0000
C01091=118.843,-37.617,32.876,-179.9780,0.1342,0.0000
C01092=117.736,-41.845,32.947,179.9855,-0.0427,0.0000
C01093=116.275,-45.866,32.994,179.9984,-0.0040,0.0000
C01094=114.651,-49.786,32.994,179.9982,-0.0040,0.0000
C01095=112.841,-53.663,32.947,179.9801,-0.0404,0.0000
C01096=110.633,-57.435,32.876,-179.9207,0.1105,0.0000
C01097=107.872,-60.637,32.806,179.2986,-0.6720,0.0000
C01098=105.013,-62.832,32.719,177.6749,-1.3092,0.0000
C01099=102.449,-63.786,32.553,175.6774,-0.9256,0.0000
C01100=99.994,-64.170,32.213,171.8839,-0.8550,0.0000
C01101=97.632,-64.599,31.757,164.9812,-3.3031,0.0000
C01102=95.273,-65.609,31.300,158.0705,-11.7512,0.0000
C01103=92.574,-67.860,30.958,157.3753,-22.2369,0.0000
C01104=89.039,-71.911,30.820,158.2381,-25.2294,0.0000
C01105=85.231,-76.357,30.814,157.5718,-24.8127,0.0000
C01106=80.918,-80.918,30.818,156.3444,-23.6551,0.0000
C01107=76.357,-85.231,30.814,155.1875,-22.4285,0.0000
C01108=71.910,-89.040,30.820,154.7711,-21.7624,0.0000
C01109=67.860,-92.574,30.958,157.7627,-22.6244,0.0000
C01110=65.609,-95.273,31.300,168.2488,-21.9295,0.0000
C01111=64.599,-97.632,31.757,176.6969,-15.0188,0.0000
C01112=64.170,-99.994,32.213,179.1450,-8.1161,0.0000
C01113=63.786,-102.449,32.553,179.0744,-4.3226,0.0000
C01114=62.832,-105.013,32.719,178.6908,-2.3251,0.0000
C01115=60.637,-107.872,32.806,179.3280,-0.7014,0.0000
C01116=57.435,-110.633,32.876,-179.8895,0.0793,0.0000
C01117=53.663,-112.841,32.947,179.9596,-0.0199,0.0000
C01118=49.786,-114.651,32.994,179.9960,-0.0018,0.0000
C01119=45.866,-116.275,32.994,179.9960,-0.0016,0.0000
C01120=41.845,-117.736,32.947,179.9573,-0.0145,0.0000
C01121=37.617,-118.843,32.876,-179.8658,0.0220,0.0000
C01122=33.400,-119.154,32.806,179.0289,0.0208,0.0000
C01123=29.826,-118.684,32.719,177.4308,0.7190,0.0000
C01124=27.339,-117.546,32.553,176.2883,2.4064,0.0000
C01125=25.331,-116.081,32.213,173.6439,5.1590,0.0000
C01126=23.358,-114.715,31.757,167.0185,8.4695,0.0000
C01127=20.976,-113.761,31.300,156.6467,7.8338,0.0000
C01128=17.476,-113.444,30.958,149.7238,0.3209,0.0000
C01129=12.112,-113.809,30.820,148.3894,-2.9141,0.0000
C01130=6.275,-114.260,30.814,148.2518,-2.0082,0.0000
C01131=0.000,-114.436,30.818,148.2225,0.0004,0.0000
C01132=0.000,-114.436,30.818,148.2225,0.0004,0.0000
C01133=-6.275,-114.260,30.814,148.2518,2.0077,0.0000
C01134=-12.112,-113.809,30.820,148.3894,2.9133,0.0000
C01135=-17.476,-113.444,30.958,149.7238,-0.3204,0.0000
C01136=-20.976,-113.761,31.300,156.6467,-7.8338,0.0000
C01137=-23.358,-114.715,31.757,167.0185,-8.4695,0.0000
C01138=-25.331,-116.081,32.213,173.6439,-5.1590,0.0000
C01139=-27.339,-117.546,32.553,176.2883,-2.4064,0.0000
C01140=-29.826,-118.684,32.719,177.4308,-0.7190,0.0000
C01141=-33.400,-119.154,32.806,179.0289,-0.0208,0.0000
C01142=-37.617,-118.843,32.876,-179.8658,-0.0220,0.0000
C01143=-41.845,-117.736,32.947,179.9573,0.0145,0.0000
C01144=-45.866,-116.275,32.994,179.9960,0.0016,0.0000
C01145=-49.786,-114.651,32.994,179.9960,0.0018,0.0000
C01146=-53.663,-112.841,32.947,179.9596,0.0199,0.0000
C01147=-57.435,-110.633,32.876,-179.8895,-0.0793,0.0000
C01148=-60.637,-107.872,32.806,179.3280,0.7014,0.0000
C01149=-62.832,-105.013,32.719,178.6908,2.3251,0.0000
C01150=-63.786,-102.449,32.553,179.0744,4.3226,0.0000
C01151=-64.170,-99.994,32.213,179.1450,8.1161,0.0000
C01152=-64.599,-97.632,31.757,176.6969,15.0188,0.0000
C01153=-65.609,-95.273,31.300,168.2488,21.9295,0.0000
C01154=-67.860,-92.574,30.958,157.7631,22.6247,0.0000
C01155=-71.911,-89.039,30.820,154.7706,21.7619,0.0000
C01156=-76.357,-85.231,30.814,155.1873,22.4282,0.0000
C01157=-80.918,-80.918,30.818,156.3449,23.6556,0.0000
C01158=-85.231,-76.357,30.814,157.5715,24.8125,0.0000
C01159=-89.040,-71.910,30.820,158.2376,25.2289,0.0000
C01160=-92.574,-67.860,30.958,157.3756,22.2373,0.0000
C01161=-95.273,-65.609,31.300,158.0705,11.7512,0.0000
C01162=-97.632,-64.599,31.757,164.9812,3.3031,0.0000
C01163=-99.994,-64.170,32.213,171.8839,0.8550,0.0000
C01164=-102.449,-63.786,32.553,175.6774,0.9256,0.0000
C01165=-105.013,-62.832,32.719,177.6749,1.3092,0.0000
C01166=-107.872,-60.637,32.806,179.2986,0.6720,0.0000
C01167=-110.633,-57.435,32.876,-179.9207,-0.1105,0.0000
C01168=-112.841,-53.663,32.947,179.9801,0.0404,0.0000
C01169=-114.651,-49.786,32.994,179.9982,0.0040,0.0000
C01170=-116.275,-45.866,32.994,179.9984,0.0040,0.0000
C01171=-117.736,-41.845,32.947,179.9855,0.0427,0.0000
C01172=-118.843,-37.617,32.876,-179.9780,-0.1342,0.0000
C01173=-119.154,-33.400,32.806,-179.9792,0.9711,0.0000
C01174=-118.684,-29.826,32.719,-179.2810,2.5692,0.0000
C01175=-117.546,-27.339,32.553,-177.5936,3.7117,0.0000
C01176=-116.081,-25.331,32.213,-174.8410,6.3561,0.0000
C01177=-114.715,-23.358,31.757,-171.5305,12.9815,0.0000
C01178=-113.761,-20.976,31.300,-172.1662,23.3533,0.0000
C01179=-113.444,-17.476,30.958,-179.6791,30.2762,0.0000
C01180=-113.809,-12.112,30.820,177.0859,31.6106,0.0000
C01181=-114.260,-6.275,30.814,177.9918,31.7482,0.0000
C01182=-114.436,0.000,30.818,-179.9996,31.7775,0.0000
C01183=-114.260,6.275,30.814,-177.9923,31.7482,0.0000
C01184=-113.809,12.112,30.820,-177.0867,31.6106,0.0000
C01185=-113.444,17.476,30.958,179.6796,30.2762,0.0000
C01186=-113.761,20.976,31.300,172.1662,23.3533,0.0000
C01187=-114.715,23.358,31.757,171.5305,12.9815,0.0000
C01188=-116.081,25.331,32.213,174.8410,6.3561,0.0000
C01189=-117.546,27.339,32.553,177.5936,3.7117,0.0000
C01190=-118.684,29.826,32.719,179.2810,2.5692,0.0000
C01191=-119.154,33.400,32.806,179.9792,0.9711,0.0000
C01192=-118.843,37.617,32.876,179.9780,-0.1342,0.0000
C01193=-117.736,41.845,32.947,-179.9855,0.0427,0.0000
C01194=-116.275,45.866,32.994,-179.9984,0.0040,0.0000
C01195=-114.651,49.786,32.994,-179.9982,0.0040,0.0000
C01196=-112.841,53.663,32.947,-179.9801,0.0404,0.0000
C01197=-110.633,57.435,32.876,179.9207,-0.1105,0.0000
C01198=-107.872,60.637,32.806,-179.2986,0.6720,0.0000
C01199=-105.013,62.832,32.719,-177.6749,1.3092,0.0000
C01200=-102.449,63.786,32.553,-175.6774,0.9256,0.0000
C01201=-99.994,64.170,32.213,-171.8839,0.8550,0.0000
C01202=-97.632,64.599,31.757,-164.9812,3.3031,0.0000
C01203=-95.273,65.609,31.300,-158.0705,11.7512,0.0000
C01204=-92.574,67.860,30.958,-157.3753,22.2369,0.0000
C01205=-89.039,71.911,30.820,-158.2381,25.2294,0.0000
C01206=-85.231,76.357,30.814,-157.5718,24.8127,0.0000
C01207=-80.918,80.918,30.818,-156.3444,23.6551,0.0000
C01208=-76.357,85.231,30.814,-155.1875,22.4285,0.0000
C01209=-71.910,89.040,30.820,-154.7711,21.7624,0.0000
C01210=-67.860,92.574,30.958,-157.7627,22.6244,0.0000
C01211=-65.609,95.273,31.300,-168.2488,21.9295,0.0000
C01212=-64.599,97.632,31.757,-176.6969,15.0188,0.0000
C01213=-64.170,99.994,32.213,-179.1450,8.1161,0.0000
C01214=-63.786,102.449,32.553,-179.0744,4.3226,0.0000
C01215=-62.832,105.013,32.719,-178.6908,2.3251,0.0000
C01216=-60.637,107.872,32.806,-179.3280,0.7014,0.0000
C01217=-57.435,110.633,32.876,179.8895,-0.0793,0.0000
C01218=-53.663,112.841,32.947,-179.9596,0.0199,0.0000
C01219=-49.786,114.651,32.994,-179.9960,0.0018,0.0000
C01220=-45.866,116.275,32.994,-179.9960,0.0016,0.0000
C01221=-41.845,117.736,32.947,-179.9573,0.0145,0.0000
C01222=-37.617,118.843,32.876,179.8658,-0.0220,0.0000
C01223=-33.400,119.154,32.806,-179.0289,-0.0208,0.0000
C01224=-29.826,118.684,32.719,-177.4308,-0.7190,0.0000
C01225=-27.339,117.546,32.553,-176.2883,-2.4064,0.0000
C01226=-25.331,116.081,32.213,-173.6439,-5.1590,0.0000
C01227=-23.358,114.715,31.757,-167.0185,-8.4695,0.0000
C01228=-20.976,113.761,31.300,-156.6467,-7.8338,0.0000
C01229=-17.476,113.444,30.958,-149.7238,-0.3204,0.0000
C01230=-12.112,113.809,30.820,-148.3894,2.9133,0.0000
C01231=-6.275,114.260,30.814,-148.2518,2.0077,0.0000
C01232=0.000,114.436,30.818,-148.2225,0.0004,0.0000
C01233=0.000,113.261,32.678,-147.2258,0.0004,0.0000
C01234=6.167,113.089,32.673,-147.2554,-2.0798,0.0000
C01235=11.931,112.648,32.680,-147.3948,-2.9034,0.0000
C01236=17.255,112.322,32.838,-148.8745,1.0288,0.0000
C01237=20.705,112.739,33.229,-157.1055,9.2308,0.0000
C01238=23.046,113.848,33.755,-168.3828,8.8098,0.0000
C01239=24.991,115.416,34.282,-174.8423,4.8516,0.0000
C01240=26.971,117.108,34.678,-177.2826,2.0776,0.0000
C01241=29.425,118.466,34.871,-178.0968,0.6631,0.0000
C01242=33.022,119.108,34.972,-179.3391,0.0366,0.0000
C01243=37.316,118.897,35.055,179.7291,0.0400,0.0000
C01244=41.655,117.799,35.138,-179.9679,-0.0108,0.0000
C01245=45.802,116.300,35.193,-179.9973,-0.0011,0.0000
C01246=49.850,114.623,35.193,-179.9973,-0.0012,0.0000
C01247=53.842,112.751,35.138,-179.9696,-0.0151,0.0000
C01248=57.687,110.460,35.055,179.7802,0.1633,0.0000
C01249=60.872,107.572,34.972,-179.5586,-0.4932,0.0000
C01250=62.961,104.575,34.871,-179.1227,-1.8145,0.0000
C01251=63.737,101.880,34.678,-179.5468,-3.3887,0.0000
C01252=63.940,99.282,34.282,-179.7819,-7.0598,0.0000
C01253=64.206,96.798,33.755,-177.9509,-14.3034,0.0000
C01254=65.078,94.359,33.229,-169.5910,-22.4666,0.0000
C01255=67.223,91.625,32.838,-157.4965,-23.7342,0.0000
C01256=71.218,88.091,32.680,-153.9799,-22.6088,0.0000
C01257=75.605,84.327,32.673,-154.3399,-23.2219,0.0000
C01258=80.087,80.087,32.678,-155.5229,-24.4776,0.0000
C01259=84.327,75.605,32.673,-156.7778,-25.6598,0.0000
C01260=88.091,71.217,32.680,-157.3907,-26.0195,0.0000
C01261=91.625,67.223,32.838,-156.2662,-22.5039,0.0000
C01262=94.359,65.078,33.229,-157.5334,-10.4090,0.0000
C01263=96.798,64.206,33.755,-165.6966,-2.0491,0.0000
C01264=99.282,63.940,34.282,-172.9402,-0.2181,0.0000
C01265=101.880,63.737,34.678,-176.6113,-0.4532,0.0000
C01266=104.575,62.961,34.871,-178.1855,-0.8773,0.0000
C01267=107.572,60.872,34.972,-179.5068,-0.4414,0.0000
C01268=110.460,57.687,35.055,179.8367,0.2198,0.0000
C01269=112.751,53.842,35.138,-179.9849,-0.0304,0.0000
C01270=114.623,49.850,35.193,-179.9988,-0.0027,0.0000
C01271=116.300,45.802,35.193,-179.9989,-0.0027,0.0000
C01272=117.799,41.655,35.138,-179.9892,-0.0321,0.0000
C01273=118.897,37.316,35.055,179.9600,0.2709,0.0000
C01274=119.108,33.022,34.972,179.9634,-0.6609,0.0000
C01275=118.466,29.425,34.871,179.3369,-1.9032,0.0000
C01276=117.108,26.971,34.678,177.9224,-2.7174,0.0000
C01277=115.416,24.991,34.282,175.1484,-5.1577,0.0000
C01278=113.848,23.046,33.755,171.1902,-11.6172,0.0000
C01279=112.739,20.705,33.229,170.7692,-22.8945,0.0000
C01280=112.322,17.255,32.838,178.9712,-31.1255,0.0000
C01281=112.648,11.931,32.680,-177.0966,-32.6052,0.0000
C01282=113.089,6.167,32.673,-177.9202,-32.7446,0.0000
C01283=113.261,0.000,32.678,179.9996,-32.7742,0.0000
C01284=113.089,-6.167,32.673,177.9207,-32.7446,0.0000
C01285=112.648,-11.931,32.680,177.0975,-32.6051,0.0000
C01286=112.322,-17.255,32.838,-178.9718,-31.1255,0.0000
C01287=112.739,-20.705,33.229,-170.7692,-22.8945,0.0000
C01288=113.848,-23.046,33.755,-171.1902,-11.6172,0.0000
C01289=115.416,-24.991,34.282,-175.1484,-5.1577,0.0000
C01290=117.108,-26.971,34.678,-177.9224,-2.7174,0.0000
C01291=118.466,-29.425,34.871,-179.3369,-1.9032,0.0000
C01292=119.108,-33.022,34.972,-179.9634,-0.6609,0.0000
C01293=118.897,-37.316,35.055,-179.9600,0.2709,0.0000
C01294=117.799,-41.655,35.138,179.9892,-0.0321,0.0000
C01295=116.300,-45.802,35.193,179.9989,-0.0027,0.0000
C01296=114.623,-49.850,35.193,179.9988,-0.0027,0.0000
C01297=112.751,-53.842,35.138,179.9849,-0.0304,0.0000
C01298=110.460,-57.687,35.055,-179.8367,0.2198,0.0000
C01299=107.572,-60.872,34.972,179.5068,-0.4414,0.0000
C01300=104.575,-62.961,34.871,178.1855,-0.8773,0.0000
C01301=101.880,-63.737,34.678,176.6113,-0.4532,0.0000
C01302=99.282,-63.940,34.282,172.9402,-0.2181,0.0000
C01303=96.798,-64.206,33.755,165.6966,-2.0491,0.0000
C01304=94.359,-65.078,33.229,157.5334,-10.4090,0.0000
C01305=91.625,-67.223,32.838,156.2658,-22.5035,0.0000
C01306=88.091,-71.218,32.680,157.3912,-26.0201,0.0000
C01307=84.327,-75.605,32.673,156.7781,-25.6601,0.0000
C01308=80.087,-80.087,32.678,155.5224,-24.4771,0.0000
C01309=75.605,-84.327,32.673,154.3402,-23.2222,0.0000
C01310=71.217,-88.091,32.680,153.9805,-22.6093,0.0000
C01311=67.223,-91.625,32.838,157.4961,-23.7338,0.0000
C01312=65.078,-94.359,33.229,169.5910,-22.4666,0.0000
C01313=64.206,-96.798,33.755,177.9509,-14.3034,0.0000
C01314=63.940,-99.282,34.282,179.7819,-7.0598,0.0000
C01315=63.737,-101.880,34.678,179.5468,-3.3887,0.0000
C01316=62.961,-104.575,34.871,179.1227,-1.8145,0.0000
C01317=60.872,-107.572,34.972,179.5586,-0.4932,0.0000
C01318=57.687,-110.460,35.055,-179.7802,0.1633,0.0000
C01319=53.842,-112.751,35.138,179.9696,-0.0151,0.0000
C01320=49.850,-114.623,35.193,179.9973,-0.0012,0.0000
C01321=45.802,-116.300,35.193,179.9973,-0.0011,0.0000
C01322=41.655,-117.799,35.138,179.9679,-0.0108,0.0000
C01323=37.316,-118.897,35.055,-179.7291,0.0400,0.0000
C01324=33.022,-119.108,34.972,179.3391,0.0366,0.0000
C01325=29.425,-118.466,34.871,178.0968,0.6631,0.0000
C01326=26.971,-117.108,34.678,177.2826,2.0776,0.0000
C01327=24.991,-115.416,34.282,174.8423,4.8516,0.0000
C01328=23.046,-113.848,33.755,168.3828,8.8098,0.0000
C01329=20.705,-112.739,33.229,157.1055,9.2308,0.0000
C01330=17.255,-112.322,32.838,148.8745,1.0288,0.0000
C01331=11.931,-112.648,32.680,147.3948,-2.9034,0.0000
C01332=6.167,-113.089,32.673,147.2554,-2.0798,0.0000
C01333=0.000,-113.261,32.678,147.2258,0.0004,0.0000
C01334=0.000,-113.261,32.678,147.2258,0.0004,0.0000
C01335=-6.167,-113.089,32.673,147.2554,2.0793,0.0000
C01336=-11.931,-112.648,32.680,147.3949,2.9025,0.0000
C01337=-17.255,-112.322,32.838,148.8745,-1.0282,0.0000
C01338=-20.705,-112.739,33.229,157.1055,-9.2308,0.0000
C01339=-23.046,-113.848,33.755,168.3828,-8.8098,0.0000
C01340=-24.991,-115.416,34.282,174.8423,-4.8516,0.0000
C01341=-26.971,-117.108,34.678,177.2826,-2.0776,0.0000
C01342=-29.425,-118.466,34.871,178.0968,-0.6631,0.0000
C01343=-33.022,-119.108,34.972,179.3391,-0.0366,0.0000
C01344=-37.316,-118.897,35.055,-179.7291,-0.0400,0.0000
C01345=-41.655,-117.799,35.138,179.9679,0.0108,0.0000
C01346=-45.802,-116.300,35.193,179.9973,0.0011,0.0000
C01347=-49.850,-114.623,35.193,179.9973,0.0012,0.0000
C01348=-53.842,-112.751,35.138,179.9696,0.0151,0.0000
C01349=-57.687,-110.460,35.055,-179.7802,-0.1633,0.0000
C01350=-60.872,-107.572,34.972,179.5586,0.4932,0.0000
C01351=-62.961,-104.575,34.871,179.1227,1.8145,0.0000
C01352=-63.737,-101.880,34.678,179.5468,3.3887,0.0000
C01353=-63.940,-99.282,34.282,179.7819,7.0598,0.0000
C01354=-64.206,-96.798,33.755,177.9509,14.3034,0.0000
C01355=-65.078,-94.359,33.229,169.5910,22.4666,0.0000
C01356=-67.223,-91.625,32.838,157.4965,23.7342,0.0000
C01357=-71.218,-88.091,32.680,153.9799,22.6088,0.0000
C01358=-75.605,-84.327,32.673,154.3399,23.2219,0.0000
C01359=-80.087,-80.087,32.678,155.5229,24.4776,0.0000
C01360=-84.327,-75.605,32.673,156.7778,25.6598,0.0000
C01361=-88.091,-71.217,32.680,157.3907,26.0195,0.0000
C01362=-91.625,-67.223,32.838,156.2662,22.5039,0.0000
C01363=-94.359,-65.078,33.229,157.5334,10.4090,0.0000
C01364=-96.798,-64.206,33.755,165.6966,2.0491,0.0000
C01365=-99.282,-63.940,34.282,172.9402,0.2181,0.0000
C01366=-101.880,-63.737,34.678,176.6113,0.4532,0.0000
C01367=-104.575,-62.961,34.871,178.1855,0.8773,0.0000
C01368=-107.572,-60.872,34.972,179.5068,0.4414,0.0000
C01369=-110.460,-57.687,35.055,-179.8367,-0.2198,0.0000
C01370=-112.751,-53.842,35.138,179.9849,0.0304,0.0000
C01371=-114.623,-49.850,35.193,179.9988,0.0027,0.0000
C01372=-116.300,-45.802,35.193,179.9989,0.0027,0.0000
C01373=-117.799,-41.655,35.138,179.9892,0.0321,0.0000
C01374=-118.897,-37.316,35.055,-179.9600,-0.2709,0.0000
C01375=-119.108,-33.022,34.972,-179.9634,0.6609,0.0000
C01376=-118.466,-29.425,34.871,-179.3369,1.9032,0.0000
C01377=-117.108,-26.971,34.678,-177.9224,2.7174,0.0000
C01378=-115.416,-24.991,34.282,-175.1484,5.1577,0.0000
C01379=-113.848,-23.046,33.755,-171.1902,11.6172,0.0000
C01380=-112.739,-20.705,33.229,-170.7692,22.8945,0.0000
C01381=-112.322,-17.255,32.838,-178.9712,31.1255,0.0000
C01382=-112.648,-11.931,32.680,177.0966,32.6052,0.0000
C01383=-113.089,-6.167,32.673,177.9202,32.7446,0.0000
C01384=-113.261,0.000,32.678,-179.9996,32.7742,0.0000
C01385=-113.089,6.167,32.673,-177.9207,32.7446,0.0000
C01386=-112.648,11.931,32.680,-177.0975,32.6051,0.0000
C01387=-112.322,17.255,32.838,178.9718,31.1255,0.0000
C01388=-112.739,20.705,33.229,170.7692,22.8945,0.0000
C01389=-113.848,23.046,33.755,171.1902,11.6172,0.0000
C01390=-115.416,24.991,34.282,175.1484,5.1577,0.0000
C01391=-117.108,26.971,34.678,177.9224,2.7174,0.0000
C01392=-118.466,29.425,34.871,179.3369,1.9032,0.0000
C01393=-119.108,33.022,34.972,179.9634,0.6609,0.0000
C01394=-118.897,37.316,35.055,179.9600,-0.2709,0.0000
C01395=-117.799,41.655,35.138,-179.9892,0.0321,0.0000
C01396=-116.300,45.802,35.193,-179.9989,0.0027,0.0000
C01397=-114.623,49.850,35.193,-179.9988,0.0027,0.0000
C01398=-112.751,53.842,35.138,-179.9849,0.0304,0.0000
C01399=-110.460,57.687,35.055,179.8367,-0.2198,0.0000
C01400=-107.572,60.872,34.972,-179.5068,0.4414,0.0000
C01401=-104.575,62.961,34.871,-178.1855,0.8773,0.0000
C01402=-101.880,63.737,34.678,-176.6113,0.4532,0.0000
C01403=-99.282,63.940,34.282,-172.9402,0.2181,0.0000
C01404=-96.798,64.206,33.755,-165.6966,2.0491,0.0000
C01405=-94.359,65.078,33.229,-157.5334,10.4090,0.0000
C01406=-91.625,67.223,32.838,-156.2658,22.5035,0.0000
C01407=-88.091,71.218,32.680,-157.3912,26.0201,0.0000
C01408=-84.327,75.605,32.673,-156.7781,25.6601,0.0000
C01409=-80.087,80.087,32.678,-155.5224,24.4771,0.0000
C01410=-75.605,84.327,32.673,-154.3402,23.2222,0.0000
C01411=-71.217,88.091,32.680,-153.9805,22.6093,0.0000
C01412=-67.223,91.625,32.838,-157.4961,23.7338,0.0000
C01413=-65.078,94.359,33.229,-169.5910,22.4666,0.0000
C01414=-64.206,96.798,33.755,-177.9509,14.3034,0.0000
C01415=-63.940,99.282,34.282,-179.7819,7.0598,0.0000
C01416=-63.737,101.880,34.678,-179.5468,3.3887,0.0000
C01417=-62.961,104.575,34.871,-179.1227,1.8145,0.0000
C01418=-60.872,107.572,34.972,-179.5586,0.4932,0.0000
C01419=-57.687,110.460,35.055,179.7802,-0.1633,0.0000
C01420=-53.842,112.751,35.138,-179.9696,0.0151,0.0000
C01421=-49.850,114.623,35.193,-179.9973,0.0012,0.0000
C01422=-45.802,116.300,35.193,-179.9973,0.0011,0.0000
C01423=-41.655,117.799,35.138,-179.9679,0.0108,0.0000
C01424=-37.316,118.897,35.055,179.7291,-0.0400,0.0000
C01425=-33.022,119.108,34.972,-179.3391,-0.0366,0.0000
C01426=-29.425,118.466,34.871,-178.0968,-0.6631,0.0000
C01427=-26.971,117.108,34.678,-177.2826,-2.0776,0.0000
C01428=-24.991,115.416,34.282,-174.8423,-4.8516,0.0000
C01429=-23.046,113.848,33.755,-168.3828,-8.8098,0.0000
C01430=-20.705,112.739,33.229,-157.1055,-9.2308,0.0000
C01431=-17.255,112.322,32.838,-148.8745,-1.0282,0.0000
C01432=-11.931,112.648,32.680,-147.3949,2.9025,0.0000
C01433=-6.167,113.089,32.673,-147.2554,2.0793,0.0000
C01434=0.000,113.261,32.678,-147.2258,0.0004,0.0000
C01435=0.000,112.055,34.518,-146.3219,0.0004,0.0000
C01436=6.057,111.887,34.513,-146.3519,-2.1448,0.0000
C01437=11.746,111.457,34.521,-146.4933,-2.8694,0.0000
C01438=17.028,111.171,34.699,-148.1460,1.8051,0.0000
C01439=20.426,111.688,35.142,-157.8460,10.4935,0.0000
C01440=22.725,112.954,35.739,-169.8053,8.8632,0.0000
C01441=24.639,114.728,36.342,-175.9597,4.3469,0.0000
C01442=26.591,116.655,36.797,-178.2253,1.5746,0.0000
C01443=29.010,118.240,37.019,-178.8077,0.5007,0.0000
C01444=32.630,119.061,37.137,-179.6782,0.0289,0.0000
C01445=37.005,118.954,37.232,179.5840,0.0546,0.0000
C01446=41.458,117.864,37.328,-179.9792,-0.0070,0.0000
C01447=45.735,116.326,37.391,-179.9986,-0.0005,0.0000
C01448=49.915,114.594,37.391,-179.9987,-0.0006,0.0000
C01449=54.027,112.657,37.328,-179.9804,-0.0098,0.0000
C01450=57.947,110.279,37.232,179.6672,0.2556,0.0000
C01451=61.116,107.261,37.137,-179.7929,-0.2479,0.0000
C01452=63.095,104.121,37.019,-179.5109,-1.1971,0.0000
C01453=63.685,101.290,36.797,-179.8584,-2.3677,0.0000
C01454=63.703,98.548,36.342,179.7820,-5.9202,0.0000
C01455=63.802,95.939,35.739,-179.0319,-13.3562,0.0000
C01456=64.532,93.419,35.142,-171.0813,-22.7275,0.0000
C01457=66.569,90.650,34.699,-157.3608,-24.7796,0.0000
C01458=70.506,87.118,34.521,-153.2709,-23.3982,0.0000
C01459=74.833,83.399,34.513,-153.5662,-23.9496,0.0000
C01460=79.235,79.235,34.518,-154.7709,-25.2296,0.0000
C01461=83.399,74.833,34.513,-156.0500,-26.4335,0.0000
C01462=87.118,70.506,34.521,-156.6013,-26.7285,0.0000
C01463=90.650,66.569,34.699,-155.2207,-22.6397,0.0000
C01464=93.419,64.532,35.142,-157.2725,-8.9187,0.0000
C01465=95.939,63.802,35.739,-166.6438,-0.9681,0.0000
C01466=98.548,63.703,36.342,-174.0798,0.2180,0.0000
C01467=101.290,63.685,36.797,-177.6323,-0.1416,0.0000
C01468=104.121,63.095,37.019,-178.8029,-0.4891,0.0000
C01469=107.261,61.116,37.137,-179.7521,-0.2071,0.0000
C01470=110.279,57.947,37.232,179.7444,0.3328,0.0000
C01471=112.657,54.027,37.328,-179.9902,-0.0196,0.0000
C01472=114.594,49.915,37.391,-179.9994,-0.0013,0.0000
C01473=116.326,45.735,37.391,-179.9995,-0.0014,0.0000
C01474=117.864,41.458,37.328,-179.9930,-0.0208,0.0000
C01475=118.954,37.005,37.232,179.9454,0.4160,0.0000
C01476=119.061,32.630,37.137,179.9711,-0.3218,0.0000
C01477=118.240,29.010,37.019,179.4993,-1.1923,0.0000
C01478=116.655,26.591,36.797,178.4254,-1.7747,0.0000
C01479=114.728,24.639,36.342,175.6531,-4.0403,0.0000
C01480=112.954,22.725,35.739,171.1368,-10.1947,0.0000
C01481=111.688,20.426,35.142,169.5065,-22.1540,0.0000
C01482=111.171,17.028,34.699,178.1949,-31.8540,0.0000
C01483=111.457,11.746,34.521,-177.1306,-33.5067,0.0000
C01484=111.887,6.057,34.513,-177.8552,-33.6481,0.0000
C01485=112.055,0.000,34.518,179.9996,-33.6781,0.0000
C01486=111.887,-6.057,34.513,177.8558,-33.6482,0.0000
C01487=111.457,-11.746,34.521,177.1316,-33.5067,0.0000
C01488=111.171,-17.028,34.699,-178.1955,-31.8541,0.0000
C01489=111.688,-20.426,35.142,-169.5065,-22.1540,0.0000
C01490=112.954,-22.725,35.739,-171.1368,-10.1947,0.0000
C01491=114.728,-24.639,36.342,-175.6531,-4.0403,0.0000
C01492=116.655,-26.591,36.797,-178.4254,-1.7747,0.0000
C01493=118.240,-29.010,37.019,-179.4993,-1.1923,0.0000
C01494=119.061,-32.630,37.137,-179.9711,-0.3218,0.0000
C01495=118.954,-37.005,37.232,-179.9454,0.4160,0.0000
C01496=117.864,-41.458,37.328,179.9930,-0.0208,0.0000
C01497=116.326,-45.735,37.391,179.9995,-0.0014,0.0000
C01498=114.594,-49.915,37.391,179.9994,-0.0013,0.0000
C01499=112.657,-54.027,37.328,179.9902,-0.0196,0.0000
C01500=110.279,-57.947,37.232,-179.7444,0.3328,0.0000
C01501=107.261,-61.116,37.137,179.7521,-0.2071,0.0000
C01502=104.121,-63.095,37.019,178.8029,-0.4891,0.0000
C01503=101.290,-63.685,36.797,177.6323,-0.1416,0.0000
C01504=98.548,-63.703,36.342,174.0798,0.2180,0.0000
C01505=95.939,-63.802,35.739,166.6438,-0.9681,0.0000
C01506=93.419,-64.532,35.142,157.2725,-8.9187,0.0000
C01507=90.650,-66.569,34.699,155.2204,-22.6392,0.0000
C01508=87.118,-70.506,34.521,156.6018,-26.7291,0.0000
C01509=83.399,-74.833,34.513,156.0504,-26.4338,0.0000
C01510=79.235,-79.235,34.518,154.7704,-25.2291,0.0000
C01511=74.833,-83.399,34.513,153.5665,-23.9500,0.0000
C01512=70.506,-87.118,34.521,153.2715,-23.3987,0.0000
C01513=66.569,-90.650,34.699,157.3603,-24.7793,0.0000
C01514=64.532,-93.419,35.142,171.0813,-22.7275,0.0000
C01515=63.802,-95.939,35.739,179.0319,-13.3562,0.0000
C01516=63.703,-98.548,36.342,-179.7820,-5.9202,0.0000
C01517=63.685,-101.290,36.797,179.8584,-2.3677,0.0000
C01518=63.095,-104.121,37.019,179.5109,-1.1971,0.0000
C01519=61.116,-107.261,37.137,179.7929,-0.2479,0.0000
C01520=57.947,-110.279,37.232,-179.6672,0.2556,0.0000
C01521=54.027,-112.657,37.328,179.9804,-0.0098,0.0000
C01522=49.915,-114.594,37.391,179.9987,-0.0006,0.0000
C01523=45.735,-116.326,37.391,179.9986,-0.0005,0.0000
C01524=41.458,-117.864,37.328,179.9792,-0.0070,0.0000
C01525=37.005,-118.954,37.232,-179.5840,0.0546,0.0000
C01526=32.630,-119.061,37.137,179.6782,0.0289,0.0000
C01527=29.010,-118.240,37.019,178.8077,0.5007,0.0000
C01528=26.591,-116.655,36.797,178.2253,1.5746,0.0000
C01529=24.639,-114.728,36.342,175.9597,4.3469,0.0000
C01530=22.725,-112.954,35.739,169.8053,8.8632,0.0000
C01531=20.426,-111.688,35.142,157.8460,10.4935,0.0000
C01532=17.028,-111.171,34.699,148.1460,1.8051,0.0000
C01533=11.746,-111.457,34.521,146.4933,-2.8694,0.0000
C01534=6.057,-111.887,34.513,146.3519,-2.1448,0.0000
C01535=0.000,-112.055,34.518,146.3219,0.0004,0.0000
C01536=0.000,-112.055,34.518,146.3219,0.0004,0.0000
C01537=-6.057,-111.887,34.513,146.3518,2.1442,0.0000
C01538=-11.746,-111.457,34.521,146.4933,2.8684,0.0000
C01539=-17.028,-111.171,34.699,148.1459,-1.8045,0.0000
C01540=-20.426,-111.688,35.142,157.8460,-10.4935,0.0000
C01541=-22.725,-112.954,35.739,169.8053,-8.8632,0.0000
C01542=-24.639,-114.728,36.342,175.9597,-4.3469,0.0000
C01543=-26.591,-116.655,36.797,178.2253,-1.5746,0.0000
C01544=-29.010,-118.240,37.019,178.8077,-0.5007,0.0000
C01545=-32.630,-119.061,37.137,179.6782,-0.0289,0.0000
C01546=-37.005,-118.954,37.232,-179.5840,-0.0546,0.0000
C01547=-41.458,-117.864,37.328,179.9792,0.0070,0.0000
C01548=-45.735,-116.326,37.391,179.9986,0.0005,0.0000
C01549=-49.915,-114.594,37.391,179.9987,0.0006,0.0000
C01550=-54.027,-112.657,37.328,179.9804,0.0098,0.0000
C01551=-57.947,-110.279,37.232,-179.6672,-0.2556,0.0000
C01552=-61.116,-107.261,37.137,179.7929,0.2479,0.0000
C01553=-63.095,-104.121,37.019,179.5109,1.1971,0.0000
C01554=-63.685,-101.290,36.797,179.8584,2.3677,0.0000
C01555=-63.703,-98.548,36.342,-179.7820,5.9202,0.0000
C01556=-63.802,-95.939,35.739,179.0319,13.3562,0.0000
C01557=-64.532,-93.419,35.142,171.0813,22.7275,0.0000
C01558=-66.569,-90.650,34.699,157.3608,24.7796,0.0000
C01559=-70.506,-87.118,34.521,153.2709,23.3982,0.0000
C01560=-74.833,-83.399,34.513,153.5662,23.9496,0.0000
C01561=-79.235,-79.235,34.518,154.7709,25.2296,0.0000
C01562=-83.399,-74.833,34.513,156.0500,26.4335,0.0000
C01563=-87.118,-70.506,34.521,156.6013,26.7285,0.0000
C01564=-90.650,-66.569,34.699,155.2207,22.6397,0.0000
C01565=-93.419,-64.532,35.142,157.2725,8.9187,0.0000
C01566=-95.939,-63.802,35.739,166.6438,0.9681,0.0000
C01567=-98.548,-63.703,36.342,174.0798,-0.2180,0.0000
C01568=-101.290,-63.685,36.797,177.6323,0.1416,0.0000
C01569=-104.121,-63.095,37.019,178.8029,0.4891,0.0000
C01570=-107.261,-61.116,37.137,179.7521,0.2071,0.0000
C01571=-110.279,-57.947,37.232,-179.7444,-0.3328,0.0000
C01572=-112.657,-54.027,37.328,179.9902,0.0196,0.0000
C01573=-114.594,-49.915,37.391,179.9994,0.0013,0.0000
C01574=-116.326,-45.735,37.391,179.9995,0.0014,0.0000
C01575=-117.864,-41.458,37.328,179.9930,0.0208,0.0000
C01576=-118.954,-37.005,37.232,-179.9454,-0.4160,0.0000
C01577=-119.061,-32.630,37.137,-179.9711,0.3218,0.0000
C01578=-118.240,-29.010,37.019,-179.4993,1.1923,0.0000
C01579=-116.655,-26.591,36.797,-178.4254,1.7747,0.0000
C01580=-114.728,-24.639,36.342,-175.6531,4.0403,0.0000
C01581=-112.954,-22.725,35.739,-171.1368,10.1947,0.0000
C01582=-111.688,-20.426,35.142,-169.5065,22.1540,0.0000
C01583=-111.171,-17.028,34.699,-178.1949,31.8540,0.0000
C01584=-111.457,-11.746,34.521,177.1306,33.5067,0.0000
C01585=-111.887,-6.057,34.513,177.8552,33.6481,0.0000
C01586=-112.055,0.000,34.518,-179.9996,33.6781,0.0000
C01587=-111.887,6.057,34.513,-177.8558,33.6482,0.0000
C01588=-111.457,11.746,34.521,-177.1316,33.5067,0.0000
C01589=-111.171,17.028,34.699,178.1955,31.8541,0.0000
C01590=-111.688,20.426,35.142,169.5065,22.1540,0.0000
C01591=-112.954,22.725,35.739,171.1368,10.1947,0.0000
C01592=-114.728,24.639,36.342,175.6531,4.0403,0.0000
C01593=-116.655,26.591,36.797,178.4254,1.7747,0.0000
C01594=-118.240,29.010,37.019,179.4993,1.1923,0.0000
C01595=-119.061,32.630,37.137,179.9711,0.3218,0.0000
C01596=-118.954,37.005,37.232,179.9454,-0.4160,0.0000
C01597=-117.864,41.458,37.328,-179.9930,0.0208,0.0000
C01598=-116.326,45.735,37.391,-179.9995,0.0014,0.0000
C01599=-114.594,49.915,37.391,-179.9994,0.0013,0.0000
C01600=-112.657,54.027,37.328,-179.9902,0.0196,0.0000
C01601=-110.279,57.947,37.232,179.7444,-0.3328,0.0000
C01602=-107.261,61.116,37.137,-179.7521,0.2071,0.0000
C01603=-104.121,63.095,37.019,-178.8029,0.4891,0.0000
C01604=-101.290,63.685,36.797,-177.6323,0.1416,0.0000
C01605=-98.548,63.703,36.342,-174.0798,-0.2180,0.0000
C01606=-95.939,63.802,35.739,-166.6438,0.9681,0.0000
C01607=-93.419,64.532,35.142,-157.2725,8.9187,0.0000
C01608=-90.650,66.569,34.699,-155.2204,22.6392,0.0000
C01609=-87.118,70.506,34.521,-156.6018,26.7291,0.0000
C01610=-83.399,74.833,34.513,-156.0504,26.4338,0.0000
C01611=-79.235,79.235,34.518,-154.7704,25.2291,0.0000
C01612=-74.833,83.399,34.513,-153.5665,23.9500,0.0000
C01613=-70.506,87.118,34.521,-153.2715,23.3987,0.0000
C01614=-66.569,90.650,34.699,-157.3603,24.7793,0.0000
C01615=-64.532,93.419,35.142,-171.0813,22.7275,0.0000
C01616=-63.802,95.939,35.739,-179.0319,13.3562,0.0000
C01617=-63.703,98.548,36.342,179.7820,5.9202,0.0000
C01618=-63.685,101.290,36.797,-179.8584,2.3677,0.0000
C01619=-63.095,104.121,37.019,-179.5109,1.1971,0.0000
C01620=-61.116,107.261,37.137,-179.7929,0.2479,0.0000
C01621=-57.947,110.279,37.232,179.6672,-0.2556,0.0000
C01622=-54.027,112.657,37.328,-179.9804,0.0098,0.0000
C01623=-49.915,114.594,37.391,-179.9987,0.0006,0.0000
C01624=-45.735,116.326,37.391,-179.9986,0.0005,0.0000
C01625=-41.458,117.864,37.328,-179.9792,0.0070,0.0000
C01626=-37.005,118.954,37.232,179.5840,-0.0546,0.0000
C01627=-32.630,119.061,37.137,-179.6782,-0.0289,0.0000
C01628=-29.010,118.240,37.019,-178.8077,-0.5007,0.0000
C01629=-26.591,116.655,36.797,-178.2253,-1.5746,0.0000
C01630=-24.639,114.728,36.342,-175.9597,-4.3469,0.0000
C01631=-22.725,112.954,35.739,-169.8053,-8.8632,0.0000
C01632=-20.426,111.688,35.142,-157.8460,-10.4935,0.0000
C01633=-17.028,111.171,34.699,-148.1459,-1.8045,0.0000
C01634=-11.746,111.457,34.521,-146.4933,2.8684,0.0000
C01635=-6.057,111.887,34.513,-146.3518,2.1442,0.0000
C01636=0.000,112.055,34.518,-146.3219,0.0004,0.0000
C01637=0.000,110.822,36.340,-145.5041,0.0004,0.0000
C01638=5.945,110.658,36.334,-145.5343,-2.2031,0.0000
C01639=11.557,110.239,36.343,-145.6782,-2.8129,0.0000
C01640=16.795,109.993,36.542,-147.5344,2.6416,0.0000
C01641=20.140,110.611,37.039,-158.8395,11.5711,0.0000
C01642=22.395,112.037,37.712,-171.2135,8.6616,0.0000
C01643=24.277,114.021,38.393,-176.9614,3.6986,0.0000
C01644=26.199,116.189,38.910,-179.0772,0.9380,0.0000
C01645=28.581,118.007,39.165,-179.5325,0.2311,0.0000
C01646=32.225,119.012,39.299,179.9614,-0.0048,0.0000
C01647=36.683,119.012,39.408,179.4325,0.0653,0.0000
C01648=41.254,117.931,39.518,-179.9911,-0.0029,0.0000
C01649=45.666,116.352,39.590,179.9999,0.0000,0.0000
C01650=49.983,114.564,39.590,179.9999,0.0000,0.0000
C01651=54.219,112.561,39.518,-179.9916,-0.0042,0.0000
C01652=58.215,110.093,39.408,179.5526,0.3551,0.0000
C01653=61.368,106.941,39.299,179.9761,0.0307,0.0000
C01654=63.233,103.653,39.165,-179.8328,-0.4940,0.0000
C01655=63.633,100.683,38.910,179.9892,-1.3157,0.0000
C01656=63.459,97.792,38.393,179.5317,-4.7586,0.0000
C01657=63.387,95.058,37.712,-179.9096,-12.2441,0.0000
C01658=63.972,92.455,37.039,-172.6533,-22.7085,0.0000
C01659=65.901,89.653,36.542,-157.3514,-25.7575,0.0000
C01660=69.779,86.123,36.343,-152.6388,-24.1328,0.0000
C01661=74.044,82.451,36.334,-152.8621,-24.6152,0.0000
C01662=78.363,78.363,36.340,-154.0849,-25.9156,0.0000
C01663=82.451,74.044,36.334,-155.3845,-27.1376,0.0000
C01664=86.123,69.779,36.343,-155.8667,-27.3605,0.0000
C01665=89.653,65.901,36.542,-154.2429,-22.6491,0.0000
C01666=92.455,63.972,37.039,-157.2915,-7.3467,0.0000
C01667=95.058,63.387,37.712,-167.7559,-0.0904,0.0000
C01668=97.792,63.459,38.393,-175.2414,0.4683,0.0000
C01669=100.683,63.633,38.910,-178.6843,0.0108,0.0000
C01670=103.653,63.233,39.165,-179.5060,-0.1672,0.0000
C01671=106.941,61.368,39.299,179.9693,0.0239,0.0000
C01672=110.093,58.215,39.408,179.6449,0.4474,0.0000
C01673=112.561,54.219,39.518,-179.9958,-0.0084,0.0000
C01674=114.564,49.983,39.590,180.0000,0.0001,0.0000
C01675=116.352,45.666,39.590,180.0000,0.0001,0.0000
C01676=117.931,41.254,39.518,-179.9971,-0.0089,0.0000
C01677=119.012,36.683,39.408,179.9347,0.5675,0.0000
C01678=119.012,32.225,39.299,-179.9952,0.0386,0.0000
C01679=118.007,28.581,39.165,179.7689,-0.4675,0.0000
C01680=116.189,26.199,38.910,179.0620,-0.9228,0.0000
C01681=114.021,24.277,38.393,176.3014,-3.0386,0.0000
C01682=112.037,22.395,37.712,171.3384,-8.7865,0.0000
C01683=110.611,20.140,37.039,168.4289,-21.1605,0.0000
C01684=109.993,16.795,36.542,177.3584,-32.4656,0.0000
C01685=110.239,11.557,36.343,-177.1871,-34.3218,0.0000
C01686=110.658,5.945,36.334,-177.7969,-34.4657,0.0000
C01687=110.822,0.000,36.340,179.9996,-34.4959,0.0000
C01688=110.659,-5.944,36.334,177.7974,-34.4658,0.0000
C01689=110.239,-11.557,36.343,177.1883,-34.3217,0.0000
C01690=109.993,-16.795,36.542,-177.3591,-32.4657,0.0000
C01691=110.611,-20.140,37.039,-168.4289,-21.1605,0.0000
C01692=112.037,-22.395,37.712,-171.3384,-8.7865,0.0000
C01693=114.021,-24.277,38.393,-176.3014,-3.0386,0.0000
C01694=116.189,-26.199,38.910,-179.0620,-0.9228,0.0000
C01695=118.007,-28.581,39.165,-179.7689,-0.4675,0.0000
C01696=119.012,-32.225,39.299,179.9952,0.0386,0.0000
C01697=119.012,-36.683,39.408,-179.9347,0.5675,0.0000
C01698=117.931,-41.254,39.518,179.9971,-0.0089,0.0000
C01699=116.352,-45.666,39.590,-180.0000,0.0001,0.0000
C01700=114.564,-49.983,39.590,-180.0000,0.0001,0.0000
C01701=112.561,-54.219,39.518,179.9958,-0.0084,0.0000
C01702=110.093,-58.215,39.408,-179.6449,0.4474,0.0000
C01703=106.941,-61.368,39.299,-179.9693,0.0239,0.0000
C01704=103.653,-63.233,39.165,179.5060,-0.1672,0.0000
C01705=100.683,-63.633,38.910,178.6843,0.0108,0.0000
C01706=97.792,-63.459,38.393,175.2414,0.4683,0.0000
C01707=95.058,-63.387,37.712,167.7559,-0.0904,0.0000
C01708=92.455,-63.972,37.039,157.2915,-7.3467,0.0000
C01709=89.653,-65.901,36.542,154.2425,-22.6486,0.0000
C01710=86.123,-69.779,36.343,155.8672,-27.3612,0.0000
C01711=82.451,-74.044,36.334,155.3848,-27.1379,0.0000
C01712=78.363,-78.363,36.340,154.0844,-25.9151,0.0000
C01713=74.044,-82.451,36.334,152.8624,-24.6155,0.0000
C01714=69.779,-86.123,36.343,152.6395,-24.1333,0.0000
C01715=65.901,-89.653,36.542,157.3509,-25.7571,0.0000
C01716=63.972,-92.455,37.039,172.6533,-22.7085,0.0000
C01717=63.387,-95.058,37.712,179.9096,-12.2441,0.0000
C01718=63.459,-97.792,38.393,-179.5317,-4.7586,0.0000
C01719=63.633,-100.683,38.910,-179.9892,-1.3157,0.0000
C01720=63.233,-103.653,39.165,179.8328,-0.4940,0.0000
C01721=61.368,-106.941,39.299,-179.9761,0.0307,0.0000
C01722=58.215,-110.093,39.408,-179.5526,0.3551,0.0000
C01723=54.219,-112.561,39.518,179.9916,-0.0042,0.0000
C01724=49.983,-114.564,39.590,-179.9999,0.0000,0.0000
C01725=45.666,-116.352,39.590,-179.9999,0.0000,0.0000
C01726=41.254,-117.931,39.518,179.9911,-0.0029,0.0000
C01727=36.683,-119.012,39.408,-179.4325,0.0653,0.0000
C01728=32.225,-119.012,39.299,-179.9614,-0.0048,0.0000
C01729=28.581,-118.007,39.165,179.5325,0.2311,0.0000
C01730=26.199,-116.189,38.910,179.0772,0.9380,0.0000
C01731=24.277,-114.021,38.393,176.9614,3.6986,0.0000
C01732=22.395,-112.037,37.712,171.2135,8.6616,0.0000
C01733=20.140,-110.611,37.039,158.8395,11.5711,0.0000
C01734=16.795,-109.993,36.542,147.5344,2.6416,0.0000
C01735=11.557,-110.239,36.343,145.6782,-2.8129,0.0000
C01736=5.945,-110.658,36.334,145.5343,-2.2031,0.0000
C01737=0.000,-110.822,36.340,145.5041,0.0004,0.0000
C01738=0.000,-110.822,36.340,145.5041,0.0004,0.0000
C01739=-5.944,-110.659,36.334,145.5342,2.2026,0.0000
C01740=-11.557,-110.239,36.343,145.6783,2.8117,0.0000
C01741=-16.795,-109.993,36.542,147.5343,-2.6409,0.0000
C01742=-20.140,-110.611,37.039,158.8395,-11.5711,0.0000
C01743=-22.395,-112.037,37.712,171.2135,-8.6616,0.0000
C01744=-24.277,-114.021,38.393,176.9614,-3.6986,0.0000
C01745=-26.199,-116.189,38.910,179.0772,-0.9380,0.0000
C01746=-28.581,-118.007,39.165,179.5325,-0.2311,0.0000
C01747=-32.225,-119.012,39.299,-179.9614,0.0048,0.0000
C01748=-36.683,-119.012,39.408,-179.4325,-0.0653,0.0000
C01749=-41.254,-117.931,39.518,179.9911,0.0029,0.0000
C01750=-45.666,-116.352,39.590,-179.9999,-0.0000,0.0000
C01751=-49.983,-114.564,39.590,-179.9999,-0.0000,0.0000
C01752=-54.219,-112.561,39.518,179.9916,0.0042,0.0000
C01753=-58.215,-110.093,39.408,-179.5526,-0.3551,0.0000
C01754=-61.368,-106.941,39.299,-179.9761,-0.0307,0.0000
C01755=-63.233,-103.653,39.165,179.8328,0.4940,0.0000
C01756=-63.633,-100.683,38.910,-179.9892,1.3157,0.0000
C01757=-63.459,-97.792,38.393,-179.5317,4.7586,0.0000
C01758=-63.387,-95.058,37.712,179.9096,12.2441,0.0000
C01759=-63.972,-92.455,37.039,172.6533,22.7085,0.0000
C01760=-65.901,-89.653,36.542,157.3514,25.7575,0.0000
C01761=-69.779,-86.123,36.343,152.6388,24.1328,0.0000
C01762=-74.044,-82.451,36.334,152.8621,24.6152,0.0000
C01763=-78.363,-78.363,36.340,154.0849,25.9156,0.0000
C01764=-82.451,-74.044,36.334,155.3845,27.1376,0.0000
C01765=-86.123,-69.779,36.343,155.8667,27.3605,0.0000
C01766=-89.653,-65.901,36.542,154.2429,22.6491,0.0000
C01767=-92.455,-63.972,37.039,157.2915,7.3467,0.0000
C01768=-95.058,-63.387,37.712,167.7559,0.0904,0.0000
C01769=-97.792,-63.459,38.393,175.2414,-0.4683,0.0000
C01770=-100.683,-63.633,38.910,178.6843,-0.0108,0.0000
C01771=-103.653,-63.233,39.165,179.5060,0.1672,0.0000
C01772=-106.941,-61.368,39.299,-179.9693,-0.0239,0.0000
C01773=-110.093,-58.215,39.408,-179.6449,-0.4474,0.0000
C01774=-112.561,-54.219,39.518,179.9958,0.0084,0.0000
C01775=-114.564,-49.983,39.590,-180.0000,-0.0001,0.0000
C01776=-116.352,-45.666,39.590,-180.0000,-0.0001,0.0000
C01777=-117.931,-41.254,39.518,179.9971,0.0089,0.0000
C01778=-119.012,-36.683,39.408,-179.9347,-0.5675,0.0000
C01779=-119.012,-32.225,39.299,179.9952,-0.0386,0.0000
C01780=-118.007,-28.581,39.165,-179.7689,0.4675,0.0000
C01781=-116.189,-26.199,38.910,-179.0620,0.9228,0.0000
C01782=-114.021,-24.277,38.393,-176.3014,3.0386,0.0000
C01783=-112.037,-22.395,37.712,-171.3384,8.7865,0.0000
C01784=-110.611,-20.140,37.039,-168.4289,21.1605,0.0000
C01785=-109.993,-16.795,36.542,-177.3584,32.4656,0.0000
C01786=-110.239,-11.557,36.343,177.1871,34.3218,0.0000
C01787=-110.658,-5.945,36.334,177.7969,34.4657,0.0000
C01788=-110.822,0.000,36.340,-179.9996,34.4959,0.0000
C01789=-110.659,5.944,36.334,-177.7974,34.4658,0.0000
C01790=-110.239,11.557,36.343,-177.1883,34.3217,0.0000
C01791=-109.993,16.795,36.542,177.3591,32.4657,0.0000
C01792=-110.611,20.140,37.039,168.4289,21.1605,0.0000
C01793=-112.037,22.395,37.712,171.3384,8.7865,0.0000
C01794=-114.021,24.277,38.393,176.3014,3.0386,0.0000
C01795=-116.189,26.199,38.910,179.0620,0.9228,0.0000
C01796=-118.007,28.581,39.165,179.7689,0.4675,0.0000
C01797=-119.012,32.225,39.299,-179.9952,-0.0386,0.0000
C01798=-119.012,36.683,39.408,179.9347,-0.5675,0.0000
C01799=-117.931,41.254,39.518,-179.9971,0.0089,0.0000
C01800=-116.352,45.666,39.590,180.0000,-0.0001,0.0000
C01801=-114.564,49.983,39.590,180.0000,-0.0001,0.0000
C01802=-112.561,54.219,39.518,-179.9958,0.0084,0.0000
C01803=-110.093,58.215,39.408,179.6449,-0.4474,0.0000
C01804=-106.941,61.368,39.299,179.9693,-0.0239,0.0000
C01805=-103.653,63.233,39.165,-179.5060,0.1672,0.0000
C01806=-100.683,63.633,38.910,-178.6843,-0.0108,0.0000
C01807=-97.792,63.459,38.393,-175.2414,-0.4683,0.0000
C01808=-95.058,63.387,37.712,-167.7559,0.0904,0.0000
C01809=-92.455,63.972,37.039,-157.2915,7.3467,0.0000
C01810=-89.653,65.901,36.542,-154.2425,22.6486,0.0000
C01811=-86.123,69.779,36.343,-155.8672,27.3612,0.0000
C01812=-82.451,74.044,36.334,-155.3848,27.1379,0.0000
C01813=-78.363,78.363,36.340,-154.0844,25.9151,0.0000
C01814=-74.044,82.451,36.334,-152.8624,24.6155,0.0000
C01815=-69.779,86.123,36.343,-152.6395,24.1333,0.0000
C01816=-65.901,89.653,36.542,-157.3509,25.7571,0.0000
C01817=-63.972,92.455,37.039,-172.6533,22.7085,0.0000
C01818=-63.387,95.058,37.712,-179.9096,12.2441,0.0000
C01819=-63.459,97.792,38.393,179.5317,4.7586,0.0000
C01820=-63.633,100.683,38.910,179.9892,1.3157,0.0000
C01821=-63.233,103.653,39.165,-179.8328,0.4940,0.0000
C01822=-61.368,106.941,39.299,179.9761,-0.0307,0.0000
C01823=-58.215,110.093,39.408,179.5526,-0.3551,0.0000
C01824=-54.219,112.561,39.518,-179.9916,0.0042,0.0000
C01825=-49.983,114.564,39.590,179.9999,-0.0000,0.0000
C01826=-45.666,116.352,39.590,179.9999,-0.0000,0.0000
C01827=-41.254,117.931,39.518,-179.9911,0.0029,0.0000
C01828=-36.683,119.012,39.408,179.4325,-0.0653,0.0000
C01829=-32.225,119.012,39.299,179.9614,0.0048,0.0000
C01830=-28.581,118.007,39.165,-179.5325,-0.2311,0.0000
C01831=-26.199,116.189,38.910,-179.0772,-0.9380,0.0000
C01832=-24.277,114.021,38.393,-176.9614,-3.6986,0.0000
C01833=-22.395,112.037,37.712,-171.2135,-8.6616,0.0000
C01834=-20.140,110.611,37.039,-158.8395,-11.5711,0.0000
C01835=-16.795,109.993,36.542,-147.5343,-2.6409,0.0000
C01836=-11.557,110.239,36.343,-145.6783,2.8117,0.0000
C01837=-5.944,110.659,36.334,-145.5342,2.2026,0.0000
C01838=0.000,110.822,36.340,-145.5041,0.0004,0.0000
C01839=0.000,109.564,38.145,-144.7664,0.0004,0.0000
C01840=5.830,109.405,38.139,-144.7966,-2.2551,0.0000
C01841=11.363,108.997,38.148,-144.9436,-2.7346,0.0000
C01842=16.558,108.791,38.370,-147.0367,3.5288,0.0000
C01843=19.849,109.511,38.921,-160.0472,12.4271,0.0000
C01844=22.057,111.099,39.673,-172.5529,8.2489,0.0000
